  MoveL 5326 to (228.65, 164.04, 78.65) mm, rotated rx 180 ry 0 rz 180 deg; joints [-145.551, -82.193, -28.272, 62.992, 39.413, -56.586]
  Call Extruder(271.49953)
  MoveL 5327 to (228.4, 164.09, 78.65) mm, rotated rx 180 ry 0 rz 180 deg; joints [-145.535, -82.158, -28.345, 62.966, 39.444, -56.545]
  MoveL 5328 to (228.4, 164.09, 78.65) mm, rotated rx 180 ry 0 rz 180 deg; joints [-145.535, -82.158, -28.345, 62.966, 39.444, -56.545]
  Call Extruder(271.63590)
  MoveL 5329 to (228.15, 164.14, 78.65) mm, rotated rx -180 ry 0 rz 180 deg; joints [-145.518, -82.122, -28.418, 62.94, 39.475, -56.503]
  MoveL 5330 to (228.15, 164.14, 78.65) mm, rotated rx -180 ry 0 rz 180 deg; joints [-145.518, -82.122, -28.418, 62.94, 39.475, -56.503]
  Call Extruder(271.77166)
  MoveL 5331 to (227.9, 164.19, 78.65) mm, rotated rx 180 ry 0 rz 180 deg; joints [-145.502, -82.086, -28.49, 62.914, 39.505, -56.463]
  MoveL 5332 to (227.9, 164.19, 78.65) mm, rotated rx 180 ry 0 rz 180 deg; joints [-145.502, -82.086, -28.49, 62.914, 39.505, -56.463]
  Call Extruder(271.90680)
  MoveL 5333 to (227.65, 164.24, 78.65) mm, rotated rx 180 ry 0 rz -180 deg; joints [-145.485, -82.051, -28.563, 62.889, 39.536, -56.422]
  MoveL 5334 to (227.65, 164.24, 78.65) mm, rotated rx 180 ry 0 rz -180 deg; joints [-145.485, -82.051, -28.563, 62.889, 39.536, -56.422]
  Call Extruder(272.04134)
  MoveL 5335 to (227.4, 164.29, 78.65) mm, rotated rx 180 ry 0 rz 180 deg; joints [-145.469, -82.016, -28.635, 62.863, 39.566, -56.382]
  MoveL 5336 to (227.4, 164.29, 78.65) mm, rotated rx 180 ry 0 rz 180 deg; joints [-145.469, -82.016, -28.635, 62.863, 39.566, -56.382]
  Call Extruder(272.17527)
  MoveL 5337 to (227.15, 164.34, 78.65) mm, rotated rx 180 ry 0 rz -180 deg; joints [-145.453, -81.98, -28.707, 62.838, 39.597, -56.341]
  MoveL 5338 to (227.15, 164.34, 78.65) mm, rotated rx 180 ry 0 rz -180 deg; joints [-145.453, -81.98, -28.707, 62.838, 39.597, -56.341]
  Call Extruder(272.32313)
  MoveL 5339 to (226.87, 164.39, 78.65) mm, rotated rx 180 ry 0 rz -180 deg; joints [-145.435, -81.94, -28.788, 62.809, 39.63, -56.295]
  MoveL 5340 to (226.87, 164.39, 78.65) mm, rotated rx 180 ry 0 rz -180 deg; joints [-145.435, -81.94, -28.788, 62.809, 39.63, -56.295]
  Call Extruder(272.48487)
  MoveL 5341 to (226.57, 164.44, 78.65) mm, rotated rx 180 ry 0 rz 180 deg; joints [-145.415, -81.896, -28.879, 62.776, 39.668, -56.244]
  MoveL 5342 to (226.57, 164.44, 78.65) mm, rotated rx 180 ry 0 rz 180 deg; joints [-145.415, -81.896, -28.879, 62.776, 39.668, -56.244]
  Call Extruder(272.64589)
  MoveL 5343 to (226.26, 164.49, 78.65) mm, rotated rx 180 ry 0 rz -180 deg; joints [-145.396, -81.851, -28.97, 62.743, 39.705, -56.192]
  MoveL 5344 to (226.26, 164.49, 78.65) mm, rotated rx 180 ry 0 rz -180 deg; joints [-145.396, -81.851, -28.97, 62.743, 39.705, -56.192]
  Call Extruder(272.80617)
  MoveL 5345 to (225.96, 164.53, 78.65) mm, rotated rx 180 ry 0 rz 180 deg; joints [-145.377, -81.807, -29.061, 62.711, 39.742, -56.141]
  MoveL 5346 to (225.96, 164.53, 78.65) mm, rotated rx 180 ry 0 rz 180 deg; joints [-145.377, -81.807, -29.061, 62.711, 39.742, -56.141]
  Call Extruder(272.96573)
  MoveL 5347 to (225.65, 164.58, 78.65) mm, rotated rx 180 ry 0 rz 180 deg; joints [-145.357, -81.763, -29.151, 62.678, 39.779, -56.09]
  MoveL 5348 to (225.65, 164.58, 78.65) mm, rotated rx 180 ry 0 rz 180 deg; joints [-145.357, -81.763, -29.151, 62.678, 39.779, -56.09]
  Call Extruder(273.12456)
  MoveL 5349 to (225.34, 164.63, 78.65) mm, rotated rx -180 ry 0 rz 180 deg; joints [-145.338, -81.719, -29.241, 62.646, 39.817, -56.039]
  MoveL 5350 to (225.34, 164.63, 78.65) mm, rotated rx -180 ry 0 rz 180 deg; joints [-145.338, -81.719, -29.241, 62.646, 39.817, -56.039]
  Call Extruder(273.30323)
  MoveL 5351 to (225, 164.68, 78.65) mm, rotated rx -180 ry 0 rz 180 deg; joints [-145.317, -81.668, -29.344, 62.608, 39.859, -55.98]
  MoveL 5352 to (225, 164.68, 78.65) mm, rotated rx -180 ry 0 rz 180 deg; joints [-145.317, -81.668, -29.344, 62.608, 39.859, -55.98]
  Call Extruder(273.50167)
  MoveL 5353 to (224.61, 164.72, 78.65) mm, rotated rx 180 ry 0 rz 180 deg; joints [-145.293, -81.611, -29.461, 62.565, 39.906, -55.913]
  MoveL 5354 to (224.61, 164.72, 78.65) mm, rotated rx 180 ry 0 rz 180 deg; joints [-145.293, -81.611, -29.461, 62.565, 39.906, -55.913]
  Call Extruder(273.69925)
  MoveL 5355 to (224.22, 164.77, 78.65) mm, rotated rx 180 ry 0 rz 180 deg; joints [-145.27, -81.554, -29.578, 62.523, 39.953, -55.846]
  MoveL 5356 to (224.22, 164.77, 78.65) mm, rotated rx 180 ry 0 rz 180 deg; joints [-145.27, -81.554, -29.578, 62.523, 39.953, -55.846]
  Call Extruder(273.89595)
  MoveL 5357 to (223.83, 164.82, 78.65) mm, rotated rx -180 ry 0 rz 180 deg; joints [-145.246, -81.497, -29.694, 62.48, 39.999, -55.78]
  MoveL 5358 to (223.83, 164.82, 78.65) mm, rotated rx -180 ry 0 rz 180 deg; joints [-145.246, -81.497, -29.694, 62.48, 39.999, -55.78]
  Call Extruder(274.09179)
  MoveL 5359 to (223.45, 164.86, 78.65) mm, rotated rx -180 ry 0 rz 180 deg; joints [-145.223, -81.44, -29.811, 62.438, 40.046, -55.713]
  MoveL 5360 to (223.45, 164.86, 78.65) mm, rotated rx -180 ry 0 rz 180 deg; joints [-145.223, -81.44, -29.811, 62.438, 40.046, -55.713]
  Call Extruder(274.38715)
  MoveL 5361 to (222.86, 164.91, 78.65) mm, rotated rx 180 ry 0 rz 180 deg; joints [-145.189, -81.352, -29.991, 62.371, 40.117, -55.609]
  MoveL 5362 to (222.86, 164.91, 78.65) mm, rotated rx 180 ry 0 rz 180 deg; joints [-145.189, -81.352, -29.991, 62.371, 40.117, -55.609]
  Call Extruder(274.68118)
  MoveL 5363 to (222.27, 164.95, 78.65) mm, rotated rx 180 ry 0 rz -180 deg; joints [-145.155, -81.264, -30.172, 62.304, 40.188, -55.505]
  MoveL 5364 to (222.27, 164.95, 78.65) mm, rotated rx 180 ry 0 rz -180 deg; joints [-145.155, -81.264, -30.172, 62.304, 40.188, -55.505]
  Call Extruder(274.97387)
  MoveL 5365 to (221.68, 165, 78.65) mm, rotated rx 180 ry 0 rz -180 deg; joints [-145.121, -81.176, -30.351, 62.238, 40.259, -55.402]
  MoveL 5366 to (221.68, 165, 78.65) mm, rotated rx 180 ry 0 rz -180 deg; joints [-145.121, -81.176, -30.351, 62.238, 40.259, -55.402]
  Call Extruder(275.54732)
  MoveL 5367 to (220.52, 165.05, 78.65) mm, rotated rx -180 ry 0 rz -180 deg; joints [-145.056, -81, -30.712, 62.101, 40.398, -55.192]
  MoveL 5368 to (220.52, 165.05, 78.65) mm, rotated rx -180 ry 0 rz -180 deg; joints [-145.056, -81, -30.712, 62.101, 40.398, -55.192]
  Call Extruder(276.26133)
  MoveL 5369 to (219.06, 165.09, 78.65) mm, rotated rx 180 ry 0 rz -180 deg; joints [-144.977, -80.78, -31.164, 61.931, 40.572, -54.93]
  Call Extruder(393.10807)
  MoveL 5370 to (-19.06, 165.09, 78.65) mm, rotated rx 180 ry 0 rz 180 deg; joints [-127.435, -60.323, -76.536, 60.813, 65.44, -36.653]
  Call Extruder(393.53667)
  MoveL 5371 to (-19.94, 165.07, 78.65) mm, rotated rx 180 ry 0 rz 180 deg; joints [-127.348, -60.28, -76.645, 60.863, 65.523, -36.622]
  MoveL 5372 to (-19.94, 165.07, 78.65) mm, rotated rx 180 ry 0 rz 180 deg; joints [-127.348, -60.28, -76.645, 60.863, 65.523, -36.622]
  Call Extruder(394.11012)
  MoveL 5373 to (-21.1, 165.02, 78.65) mm, rotated rx 180 ry 0 rz -180 deg; joints [-127.235, -60.221, -76.793, 60.928, 65.634, -36.579]
  MoveL 5374 to (-21.1, 165.02, 78.65) mm, rotated rx 180 ry 0 rz -180 deg; joints [-127.235, -60.221, -76.793, 60.928, 65.634, -36.579]
  Call Extruder(394.54442)
  MoveL 5375 to (-21.97, 164.98, 78.65) mm, rotated rx 180 ry 0 rz -180 deg; joints [-127.15, -60.176, -76.906, 60.976, 65.718, -36.544]
  MoveL 5376 to (-21.97, 164.98, 78.65) mm, rotated rx 180 ry 0 rz -180 deg; joints [-127.15, -60.176, -76.906, 60.976, 65.718, -36.544]
  Call Extruder(394.83845)
  MoveL 5377 to (-22.56, 164.93, 78.65) mm, rotated rx 180 ry 0 rz 180 deg; joints [-127.093, -60.144, -76.984, 61.007, 65.774, -36.519]
  MoveL 5378 to (-22.56, 164.93, 78.65) mm, rotated rx 180 ry 0 rz 180 deg; joints [-127.093, -60.144, -76.984, 61.007, 65.774, -36.519]
  Call Extruder(395.13381)
  MoveL 5379 to (-23.15, 164.89, 78.65) mm, rotated rx -180 ry 0 rz -180 deg; joints [-127.037, -60.113, -77.062, 61.038, 65.83, -36.495]
  MoveL 5380 to (-23.15, 164.89, 78.65) mm, rotated rx -180 ry 0 rz -180 deg; joints [-127.037, -60.113, -77.062, 61.038, 65.83, -36.495]
  Call Extruder(395.38003)
  MoveL 5381 to (-23.64, 164.84, 78.65) mm, rotated rx 180 ry 0 rz 180 deg; joints [-126.991, -60.087, -77.128, 61.063, 65.877, -36.473]
  MoveL 5382 to (-23.64, 164.84, 78.65) mm, rotated rx 180 ry 0 rz 180 deg; joints [-126.991, -60.087, -77.128, 61.063, 65.877, -36.473]
  Call Extruder(395.57673)
  MoveL 5383 to (-24.03, 164.79, 78.65) mm, rotated rx 180 ry 0 rz 180 deg; joints [-126.955, -60.066, -77.181, 61.082, 65.914, -36.455]
  MoveL 5384 to (-24.03, 164.79, 78.65) mm, rotated rx 180 ry 0 rz 180 deg; joints [-126.955, -60.066, -77.181, 61.082, 65.914, -36.455]
  Call Extruder(395.77431)
  MoveL 5385 to (-24.42, 164.75, 78.65) mm, rotated rx 180 ry 0 rz 180 deg; joints [-126.919, -60.045, -77.235, 61.101, 65.951, -36.437]
  MoveL 5386 to (-24.42, 164.75, 78.65) mm, rotated rx 180 ry 0 rz 180 deg; joints [-126.919, -60.045, -77.235, 61.101, 65.951, -36.437]
  Call Extruder(395.97275)
  MoveL 5387 to (-24.8, 164.7, 78.65) mm, rotated rx -180 ry 0 rz 180 deg; joints [-126.883, -60.023, -77.289, 61.121, 65.988, -36.419]
  MoveL 5388 to (-24.8, 164.7, 78.65) mm, rotated rx -180 ry 0 rz 180 deg; joints [-126.883, -60.023, -77.289, 61.121, 65.988, -36.419]
  Call Extruder(396.17206)
  MoveL 5389 to (-25.19, 164.66, 78.65) mm, rotated rx 180 ry 0 rz -180 deg; joints [-126.847, -60.002, -77.342, 61.14, 66.025, -36.401]
  MoveL 5390 to (-25.19, 164.66, 78.65) mm, rotated rx 180 ry 0 rz -180 deg; joints [-126.847, -60.002, -77.342, 61.14, 66.025, -36.401]
  Call Extruder(396.33089)
  MoveL 5391 to (-25.5, 164.61, 78.65) mm, rotated rx 180 ry 0 rz 180 deg; joints [-126.82, -59.985, -77.386, 61.154, 66.054, -36.386]
  MoveL 5392 to (-25.5, 164.61, 78.65) mm, rotated rx 180 ry 0 rz 180 deg; joints [-126.82, -59.985, -77.386, 61.154, 66.054, -36.386]
  Call Extruder(396.49045)
  MoveL 5393 to (-25.8, 164.56, 78.65) mm, rotated rx -180 ry 0 rz 180 deg; joints [-126.792, -59.967, -77.43, 61.168, 66.083, -36.37]
  MoveL 5394 to (-25.8, 164.56, 78.65) mm, rotated rx -180 ry 0 rz 180 deg; joints [-126.792, -59.967, -77.43, 61.168, 66.083, -36.37]
  Call Extruder(396.65073)
  MoveL 5395 to (-26.11, 164.51, 78.65) mm, rotated rx 180 ry 0 rz 180 deg; joints [-126.765, -59.95, -77.474, 61.182, 66.112, -36.355]
  MoveL 5396 to (-26.11, 164.51, 78.65) mm, rotated rx 180 ry 0 rz 180 deg; joints [-126.765, -59.95, -77.474, 61.182, 66.112, -36.355]
  Call Extruder(396.81175)
  MoveL 5397 to (-26.41, 164.46, 78.65) mm, rotated rx -180 ry 0 rz -180 deg; joints [-126.737, -59.932, -77.518, 61.196, 66.141, -36.339]
  MoveL 5398 to (-26.41, 164.46, 78.65) mm, rotated rx -180 ry 0 rz -180 deg; joints [-126.737, -59.932, -77.518, 61.196, 66.141, -36.339]
  Call Extruder(396.97349)
  MoveL 5399 to (-26.72, 164.41, 78.65) mm, rotated rx -180 ry 0 rz 180 deg; joints [-126.71, -59.915, -77.562, 61.21, 66.17, -36.323]
  MoveL 5400 to (-26.72, 164.41, 78.65) mm, rotated rx -180 ry 0 rz 180 deg; joints [-126.71, -59.915, -77.562, 61.21, 66.17, -36.323]
  Call Extruder(397.13596)
  MoveL 5401 to (-27.03, 164.36, 78.65) mm, rotated rx -180 ry 0 rz 180 deg; joints [-126.682, -59.897, -77.606, 61.224, 66.199, -36.308]
  MoveL 5402 to (-27.03, 164.36, 78.65) mm, rotated rx -180 ry 0 rz 180 deg; joints [-126.682, -59.897, -77.606, 61.224, 66.199, -36.308]
  Call Extruder(397.26988)
  MoveL 5403 to (-27.27, 164.32, 78.65) mm, rotated rx 180 ry 0 rz -180 deg; joints [-126.66, -59.883, -77.643, 61.234, 66.223, -36.294]
  MoveL 5404 to (-27.27, 164.32, 78.65) mm, rotated rx 180 ry 0 rz -180 deg; joints [-126.66, -59.883, -77.643, 61.234, 66.223, -36.294]
  Call Extruder(397.40442)
  MoveL 5405 to (-27.52, 164.27, 78.65) mm, rotated rx 180 ry 0 rz -180 deg; joints [-126.638, -59.868, -77.68, 61.245, 66.247, -36.28]
  MoveL 5406 to (-27.52, 164.27, 78.65) mm, rotated rx 180 ry 0 rz -180 deg; joints [-126.638, -59.868, -77.68, 61.245, 66.247, -36.28]
  Call Extruder(397.53957)
  MoveL 5407 to (-27.77, 164.22, 78.65) mm, rotated rx -180 ry 0 rz 180 deg; joints [-126.617, -59.853, -77.718, 61.255, 66.271, -36.266]
  MoveL 5408 to (-27.77, 164.22, 78.65) mm, rotated rx -180 ry 0 rz 180 deg; joints [-126.617, -59.853, -77.718, 61.255, 66.271, -36.266]
  Call Extruder(397.67532)
  MoveL 5409 to (-28.02, 164.17, 78.65) mm, rotated rx -180 ry 0 rz -180 deg; joints [-126.595, -59.838, -77.755, 61.266, 66.294, -36.253]
  MoveL 5410 to (-28.02, 164.17, 78.65) mm, rotated rx -180 ry 0 rz -180 deg; joints [-126.595, -59.838, -77.755, 61.266, 66.294, -36.253]
  Call Extruder(397.81169)
  MoveL 5411 to (-28.27, 164.12, 78.65) mm, rotated rx 180 ry 0 rz 180 deg; joints [-126.573, -59.824, -77.792, 61.276, 66.318, -36.239]
  MoveL 5412 to (-28.27, 164.12, 78.65) mm, rotated rx 180 ry 0 rz 180 deg; joints [-126.573, -59.824, -77.792, 61.276, 66.318, -36.239]
  Call Extruder(397.89656)
  MoveL 5413 to (-28.42, 164.09, 78.65) mm, rotated rx 180 ry 0 rz 180 deg; joints [-126.559, -59.815, -77.815, 61.283, 66.333, -36.23]
  Set speed (130.0 mm/s)
  MoveL 5414 to (-31.76, 163.31, 78.65) mm, rotated rx 180 ry 0 rz 180 deg; joints [-126.274, -59.612, -78.328, 61.416, 66.65, -36.033]
  MoveL 5415 to (-31.76, 163.31, 88.06) mm, rotated rx 180 ry 0 rz 180 deg; joints [-126.274, -58.332, -78.939, 61.672, 66.331, -36.675]
  Call Extruder(395.89656)
  Set speed (40.0 mm/s)
  MoveL 5416 to (-31.76, 163.31, 88.06) mm, rotated rx 180 ry 0 rz 180 deg; joints [-126.274, -58.332, -78.939, 61.672, 66.331, -36.675]
  Call Extruder(0.00000)
  Set speed (130.0 mm/s)
  MoveL 5417 to (-31.64, 163.21, 88.06) mm, rotated rx 180 ry 0 rz 180 deg; joints [-126.294, -58.331, -78.941, 61.654, 66.319, -36.667]
  Call Extruder(2.00000)
  Set speed (40.0 mm/s)
  MoveL 5418 to (-31.64, 163.21, 88.06) mm, rotated rx 180 ry 0 rz 180 deg; joints [-126.294, -58.331, -78.941, 61.654, 66.319, -36.667]
  Set speed (30.0 mm/s)
  MoveL 5419 to (-31.64, 163.21, 88.06) mm, rotated rx 180 ry 0 rz 180 deg; joints [-126.294, -58.331, -78.941, 61.654, 66.319, -36.667]
  Call Extruder(2.18198)
  MoveL 5420 to (-31.93, 163.09, 88.06) mm, rotated rx -180 ry 0 rz 180 deg; joints [-126.273, -58.309, -78.994, 61.66, 66.347, -36.644]
  MoveL 5421 to (-31.93, 163.09, 88.06) mm, rotated rx -180 ry 0 rz 180 deg; joints [-126.273, -58.309, -78.994, 61.66, 66.347, -36.644]
  Call Extruder(2.36471)
  MoveL 5422 to (-32.22, 162.96, 88.06) mm, rotated rx -180 ry 0 rz 180 deg; joints [-126.252, -58.288, -79.047, 61.666, 66.375, -36.621]
  MoveL 5423 to (-32.22, 162.96, 88.06) mm, rotated rx -180 ry 0 rz 180 deg; joints [-126.252, -58.288, -79.047, 61.666, 66.375, -36.621]
  Call Extruder(2.53513)
  MoveL 5424 to (-32.49, 162.85, 88.06) mm, rotated rx 180 ry 0 rz 180 deg; joints [-126.233, -58.268, -79.097, 61.672, 66.4, -36.599]
  MoveL 5425 to (-32.49, 162.85, 88.06) mm, rotated rx 180 ry 0 rz 180 deg; joints [-126.233, -58.268, -79.097, 61.672, 66.4, -36.599]
  Call Extruder(2.69310)
  MoveL 5426 to (-32.74, 162.74, 88.06) mm, rotated rx 180 ry 0 rz 180 deg; joints [-126.215, -58.25, -79.142, 61.677, 66.424, -36.579]
  MoveL 5427 to (-32.74, 162.74, 88.06) mm, rotated rx 180 ry 0 rz 180 deg; joints [-126.215, -58.25, -79.142, 61.677, 66.424, -36.579]
  Call Extruder(2.85168)
  MoveL 5428 to (-32.99, 162.64, 88.06) mm, rotated rx 180 ry 0 rz -180 deg; joints [-126.197, -58.231, -79.188, 61.682, 66.448, -36.559]
  MoveL 5429 to (-32.99, 162.64, 88.06) mm, rotated rx 180 ry 0 rz -180 deg; joints [-126.197, -58.231, -79.188, 61.682, 66.448, -36.559]
  Call Extruder(3.05785)
  MoveL 5430 to (-33.29, 162.46, 88.06) mm, rotated rx 180 ry 0 rz 180 deg; joints [-126.179, -58.206, -79.251, 61.684, 66.476, -36.529]
  MoveL 5431 to (-33.29, 162.46, 88.06) mm, rotated rx 180 ry 0 rz 180 deg; joints [-126.179, -58.206, -79.251, 61.684, 66.476, -36.529]
  Call Extruder(3.26479)
  MoveL 5432 to (-33.6, 162.29, 88.06) mm, rotated rx 180 ry 0 rz 180 deg; joints [-126.16, -58.181, -79.314, 61.685, 66.505, -36.499]
  MoveL 5433 to (-33.6, 162.29, 88.06) mm, rotated rx 180 ry 0 rz 180 deg; joints [-126.16, -58.181, -79.314, 61.685, 66.505, -36.499]
  Call Extruder(3.47251)
  MoveL 5434 to (-33.9, 162.11, 88.06) mm, rotated rx 180 ry 0 rz 180 deg; joints [-126.142, -58.156, -79.377, 61.687, 66.534, -36.47]
  MoveL 5435 to (-33.9, 162.11, 88.06) mm, rotated rx 180 ry 0 rz 180 deg; joints [-126.142, -58.156, -79.377, 61.687, 66.534, -36.47]
  Call Extruder(3.68102)
  MoveL 5436 to (-34.21, 161.94, 88.06) mm, rotated rx 180 ry 0 rz 180 deg; joints [-126.123, -58.131, -79.44, 61.689, 66.563, -36.44]
  MoveL 5437 to (-34.21, 161.94, 88.06) mm, rotated rx 180 ry 0 rz 180 deg; joints [-126.123, -58.131, -79.44, 61.689, 66.563, -36.44]
  Call Extruder(3.86055)
  MoveL 5438 to (-34.45, 161.76, 88.06) mm, rotated rx 180 ry 0 rz 180 deg; joints [-126.111, -58.108, -79.496, 61.687, 66.586, -36.412]
  MoveL 5439 to (-34.45, 161.76, 88.06) mm, rotated rx 180 ry 0 rz 180 deg; joints [-126.111, -58.108, -79.496, 61.687, 66.586, -36.412]
  Call Extruder(4.19399)
  MoveL 5440 to (-34.9, 161.43, 88.06) mm, rotated rx 180 ry 0 rz -180 deg; joints [-126.089, -58.067, -79.6, 61.682, 66.629, -36.36]
  MoveL 5441 to (-34.9, 161.43, 88.06) mm, rotated rx 180 ry 0 rz -180 deg; joints [-126.089, -58.067, -79.6, 61.682, 66.629, -36.36]
  Call Extruder(4.52861)
  MoveL 5442 to (-35.35, 161.1, 88.06) mm, rotated rx -180 ry 0 rz 180 deg; joints [-126.067, -58.025, -79.703, 61.678, 66.672, -36.308]
  Call Extruder(5.35652)
  MoveL 5443 to (-36.39, 160.19, 88.06) mm, rotated rx 180 ry 0 rz 180 deg; joints [-126.027, -57.921, -79.966, 61.653, 66.77, -36.17]
  Call Extruder(6.18445)
  MoveL 5444 to (-37.3, 159.15, 88.06) mm, rotated rx 180 ry 0 rz 180 deg; joints [-126.011, -57.814, -80.233, 61.607, 66.856, -36.022]
  Call Extruder(6.35176)
  MoveL 5445 to (-37.47, 158.93, 88.06) mm, rotated rx -180 ry 0 rz 180 deg; joints [-126.011, -57.793, -80.288, 61.595, 66.872, -35.991]
  MoveL 5446 to (-37.47, 158.93, 88.06) mm, rotated rx -180 ry 0 rz 180 deg; joints [-126.011, -57.793, -80.288, 61.595, 66.872, -35.991]
  Call Extruder(6.68519)
  MoveL 5447 to (-37.79, 158.48, 88.06) mm, rotated rx -180 ry 0 rz 180 deg; joints [-126.011, -57.75, -80.396, 61.57, 66.903, -35.928]
  MoveL 5448 to (-37.79, 158.48, 88.06) mm, rotated rx -180 ry 0 rz 180 deg; joints [-126.011, -57.75, -80.396, 61.57, 66.903, -35.928]
  Call Extruder(7.01743)
  MoveL 5449 to (-38.12, 158.03, 88.06) mm, rotated rx 180 ry 0 rz 180 deg; joints [-126.011, -57.707, -80.504, 61.546, 66.934, -35.866]
  MoveL 5450 to (-38.12, 158.03, 88.06) mm, rotated rx 180 ry 0 rz 180 deg; joints [-126.011, -57.707, -80.504, 61.546, 66.934, -35.866]
  Call Extruder(7.13510)
  MoveL 5451 to (-38.22, 157.85, 88.06) mm, rotated rx -180 ry 0 rz 180 deg; joints [-126.013, -57.692, -80.542, 61.535, 66.943, -35.843]
  MoveL 5452 to (-38.22, 157.85, 88.06) mm, rotated rx -180 ry 0 rz 180 deg; joints [-126.013, -57.692, -80.542, 61.535, 66.943, -35.843]
  Call Extruder(7.34283)
  MoveL 5453 to (-38.4, 157.55, 88.06) mm, rotated rx -180 ry 0 rz -180 deg; joints [-126.018, -57.665, -80.61, 61.515, 66.96, -35.802]
  MoveL 5454 to (-38.4, 157.55, 88.06) mm, rotated rx -180 ry 0 rz -180 deg; joints [-126.018, -57.665, -80.61, 61.515, 66.96, -35.802]
  Call Extruder(7.54978)
  MoveL 5455 to (-38.57, 157.25, 88.06) mm, rotated rx 180 ry 0 rz 180 deg; joints [-126.023, -57.638, -80.677, 61.496, 66.976, -35.762]
  MoveL 5456 to (-38.57, 157.25, 88.06) mm, rotated rx 180 ry 0 rz 180 deg; joints [-126.023, -57.638, -80.677, 61.496, 66.976, -35.762]
  Call Extruder(7.75595)
  MoveL 5457 to (-38.75, 156.94, 88.06) mm, rotated rx -180 ry 0 rz 180 deg; joints [-126.028, -57.611, -80.745, 61.476, 66.993, -35.721]
  MoveL 5458 to (-38.75, 156.94, 88.06) mm, rotated rx -180 ry 0 rz 180 deg; joints [-126.028, -57.611, -80.745, 61.476, 66.993, -35.721]
  Call Extruder(7.93763)
  MoveL 5459 to (-38.89, 156.66, 88.06) mm, rotated rx -180 ry 0 rz 180 deg; joints [-126.034, -57.588, -80.804, 61.457, 67.006, -35.685]
  MoveL 5460 to (-38.89, 156.66, 88.06) mm, rotated rx -180 ry 0 rz 180 deg; joints [-126.034, -57.588, -80.804, 61.457, 67.006, -35.685]
  Call Extruder(8.09561)
  MoveL 5461 to (-39, 156.42, 88.06) mm, rotated rx -180 ry 0 rz 180 deg; joints [-126.042, -57.568, -80.855, 61.439, 67.017, -35.653]
  MoveL 5462 to (-39, 156.42, 88.06) mm, rotated rx -180 ry 0 rz 180 deg; joints [-126.042, -57.568, -80.855, 61.439, 67.017, -35.653]
  Call Extruder(8.25300)
  MoveL 5463 to (-39.1, 156.17, 88.06) mm, rotated rx -180 ry 0 rz -180 deg; joints [-126.05, -57.547, -80.906, 61.42, 67.027, -35.62]
  MoveL 5464 to (-39.1, 156.17, 88.06) mm, rotated rx -180 ry 0 rz -180 deg; joints [-126.05, -57.547, -80.906, 61.42, 67.027, -35.62]
  Call Extruder(8.43571)
  MoveL 5465 to (-39.23, 155.87, 88.06) mm, rotated rx -180 ry 0 rz -180 deg; joints [-126.06, -57.524, -80.966, 61.398, 67.038, -35.583]
  MoveL 5466 to (-39.23, 155.87, 88.06) mm, rotated rx -180 ry 0 rz -180 deg; joints [-126.06, -57.524, -80.966, 61.398, 67.038, -35.583]
  Call Extruder(8.61768)
  MoveL 5467 to (-39.35, 155.58, 88.06) mm, rotated rx -180 ry 0 rz 180 deg; joints [-126.07, -57.501, -81.025, 61.376, 67.05, -35.545]
  MoveL 5468 to (-39.35, 155.58, 88.06) mm, rotated rx -180 ry 0 rz 180 deg; joints [-126.07, -57.501, -81.025, 61.376, 67.05, -35.545]
  Call Extruder(8.76501)
  MoveL 5469 to (-39.44, 155.34, 88.06) mm, rotated rx 180 ry 0 rz 180 deg; joints [-126.079, -57.482, -81.073, 61.358, 67.058, -35.515]
  MoveL 5470 to (-39.44, 155.34, 88.06) mm, rotated rx 180 ry 0 rz 180 deg; joints [-126.079, -57.482, -81.073, 61.358, 67.058, -35.515]
  Call Extruder(8.87824)
  MoveL 5471 to (-39.5, 155.15, 88.06) mm, rotated rx -180 ry 0 rz 180 deg; joints [-126.087, -57.467, -81.109, 61.342, 67.064, -35.491]
  MoveL 5472 to (-39.5, 155.15, 88.06) mm, rotated rx -180 ry 0 rz 180 deg; joints [-126.087, -57.467, -81.109, 61.342, 67.064, -35.491]
  Call Extruder(8.99103)
  MoveL 5473 to (-39.56, 154.97, 88.06) mm, rotated rx -180 ry 0 rz 180 deg; joints [-126.095, -57.453, -81.145, 61.327, 67.07, -35.467]
  MoveL 5474 to (-39.56, 154.97, 88.06) mm, rotated rx -180 ry 0 rz 180 deg; joints [-126.095, -57.453, -81.145, 61.327, 67.07, -35.467]
  Call Extruder(9.10338)
  MoveL 5475 to (-39.62, 154.78, 88.06) mm, rotated rx -180 ry 0 rz 180 deg; joints [-126.103, -57.439, -81.182, 61.312, 67.076, -35.443]
  MoveL 5476 to (-39.62, 154.78, 88.06) mm, rotated rx -180 ry 0 rz 180 deg; joints [-126.103, -57.439, -81.182, 61.312, 67.076, -35.443]
  Call Extruder(9.21528)
  MoveL 5477 to (-39.68, 154.59, 88.06) mm, rotated rx 180 ry 0 rz 180 deg; joints [-126.111, -57.425, -81.218, 61.296, 67.082, -35.42]
  MoveL 5478 to (-39.68, 154.59, 88.06) mm, rotated rx 180 ry 0 rz 180 deg; joints [-126.111, -57.425, -81.218, 61.296, 67.082, -35.42]
  Call Extruder(9.33668)
  MoveL 5479 to (-39.75, 154.38, 88.06) mm, rotated rx -180 ry 0 rz 180 deg; joints [-126.12, -57.409, -81.257, 61.279, 67.088, -35.394]
  MoveL 5480 to (-39.75, 154.38, 88.06) mm, rotated rx -180 ry 0 rz 180 deg; joints [-126.12, -57.409, -81.257, 61.279, 67.088, -35.394]
  Call Extruder(9.46747)
  MoveL 5481 to (-39.82, 154.16, 88.06) mm, rotated rx -180 ry 0 rz 180 deg; joints [-126.131, -57.392, -81.3, 61.261, 67.094, -35.366]
  MoveL 5482 to (-39.82, 154.16, 88.06) mm, rotated rx -180 ry 0 rz 180 deg; joints [-126.131, -57.392, -81.3, 61.261, 67.094, -35.366]
  Call Extruder(9.59770)
  MoveL 5483 to (-39.88, 153.94, 88.06) mm, rotated rx 180 ry 0 rz -180 deg; joints [-126.141, -57.376, -81.342, 61.242, 67.101, -35.338]
  MoveL 5484 to (-39.88, 153.94, 88.06) mm, rotated rx 180 ry 0 rz -180 deg; joints [-126.141, -57.376, -81.342, 61.242, 67.101, -35.338]
  Call Extruder(9.72737)
  MoveL 5485 to (-39.95, 153.71, 88.06) mm, rotated rx 180 ry 0 rz 180 deg; joints [-126.151, -57.359, -81.384, 61.223, 67.107, -35.31]
  MoveL 5486 to (-39.95, 153.71, 88.06) mm, rotated rx 180 ry 0 rz 180 deg; joints [-126.151, -57.359, -81.384, 61.223, 67.107, -35.31]
  Call Extruder(9.85647)
  MoveL 5487 to (-40.02, 153.49, 88.06) mm, rotated rx 180 ry 0 rz -180 deg; joints [-126.161, -57.342, -81.427, 61.205, 67.113, -35.282]
  MoveL 5488 to (-40.02, 153.49, 88.06) mm, rotated rx 180 ry 0 rz -180 deg; joints [-126.161, -57.342, -81.427, 61.205, 67.113, -35.282]
  Call Extruder(9.97156)
  MoveL 5489 to (-40.06, 153.28, 88.06) mm, rotated rx -180 ry 0 rz 180 deg; joints [-126.173, -57.328, -81.463, 61.187, 67.118, -35.257]
  MoveL 5490 to (-40.06, 153.28, 88.06) mm, rotated rx -180 ry 0 rz 180 deg; joints [-126.173, -57.328, -81.463, 61.187, 67.118, -35.257]
  Call Extruder(10.08619)
  MoveL 5491 to (-40.11, 153.08, 88.06) mm, rotated rx 180 ry 0 rz 180 deg; joints [-126.184, -57.313, -81.5, 61.169, 67.122, -35.232]
  MoveL 5492 to (-40.11, 153.08, 88.06) mm, rotated rx 180 ry 0 rz 180 deg; joints [-126.184, -57.313, -81.5, 61.169, 67.122, -35.232]
  Call Extruder(10.20038)
  MoveL 5493 to (-40.15, 152.88, 88.06) mm, rotated rx 180 ry 0 rz 180 deg; joints [-126.195, -57.299, -81.537, 61.15, 67.126, -35.207]
  MoveL 5494 to (-40.15, 152.88, 88.06) mm, rotated rx 180 ry 0 rz 180 deg; joints [-126.195, -57.299, -81.537, 61.15, 67.126, -35.207]
  Call Extruder(10.31411)
  MoveL 5495 to (-40.2, 152.67, 88.06) mm, rotated rx 180 ry 0 rz 180 deg; joints [-126.206, -57.285, -81.574, 61.132, 67.13, -35.182]
  MoveL 5496 to (-40.2, 152.67, 88.06) mm, rotated rx 180 ry 0 rz 180 deg; joints [-126.206, -57.285, -81.574, 61.132, 67.13, -35.182]
  Call Extruder(10.43953)
  MoveL 5497 to (-40.24, 152.45, 88.06) mm, rotated rx 180 ry 0 rz 180 deg; joints [-126.219, -57.269, -81.614, 61.112, 67.135, -35.154]
  MoveL 5498 to (-40.24, 152.45, 88.06) mm, rotated rx 180 ry 0 rz 180 deg; joints [-126.219, -57.269, -81.614, 61.112, 67.135, -35.154]
  Call Extruder(10.57651)
  MoveL 5499 to (-40.29, 152.19, 88.06) mm, rotated rx -180 ry 0 rz 180 deg; joints [-126.233, -57.251, -81.658, 61.089, 67.14, -35.123]
  MoveL 5500 to (-40.29, 152.19, 88.06) mm, rotated rx -180 ry 0 rz 180 deg; joints [-126.233, -57.251, -81.658, 61.089, 67.14, -35.123]
  Call Extruder(10.71287)
  MoveL 5501 to (-40.34, 151.95, 88.06) mm, rotated rx 180 ry 0 rz 180 deg; joints [-126.248, -57.234, -81.702, 61.066, 67.144, -35.093]
  MoveL 5502 to (-40.34, 151.95, 88.06) mm, rotated rx 180 ry 0 rz 180 deg; joints [-126.248, -57.234, -81.702, 61.066, 67.144, -35.093]
  Call Extruder(10.84863)
  MoveL 5503 to (-40.39, 151.7, 88.06) mm, rotated rx 180 ry 0 rz 180 deg; joints [-126.262, -57.217, -81.746, 61.044, 67.149, -35.063]
  MoveL 5504 to (-40.39, 151.7, 88.06) mm, rotated rx 180 ry 0 rz 180 deg; joints [-126.262, -57.217, -81.746, 61.044, 67.149, -35.063]
  Call Extruder(10.98377)
  MoveL 5505 to (-40.44, 151.45, 88.06) mm, rotated rx -180 ry 0 rz 180 deg; joints [-126.276, -57.199, -81.79, 61.021, 67.154, -35.032]
  MoveL 5506 to (-40.44, 151.45, 88.06) mm, rotated rx -180 ry 0 rz 180 deg; joints [-126.276, -57.199, -81.79, 61.021, 67.154, -35.032]
  Call Extruder(11.11831)
  MoveL 5507 to (-40.49, 151.2, 88.06) mm, rotated rx -180 ry 0 rz -180 deg; joints [-126.291, -57.182, -81.834, 60.999, 67.159, -35.002]
  MoveL 5508 to (-40.49, 151.2, 88.06) mm, rotated rx -180 ry 0 rz -180 deg; joints [-126.291, -57.182, -81.834, 60.999, 67.159, -35.002]
  Call Extruder(11.25223)
  MoveL 5509 to (-40.54, 150.95, 88.06) mm, rotated rx 180 ry 0 rz 180 deg; joints [-126.305, -57.165, -81.878, 60.976, 67.163, -34.972]
  MoveL 5510 to (-40.54, 150.95, 88.06) mm, rotated rx 180 ry 0 rz 180 deg; joints [-126.305, -57.165, -81.878, 60.976, 67.163, -34.972]
  Call Extruder(11.40009)
  MoveL 5511 to (-40.59, 150.67, 88.06) mm, rotated rx -180 ry 0 rz 180 deg; joints [-126.322, -57.146, -81.927, 60.95, 67.168, -34.938]
  MoveL 5512 to (-40.59, 150.67, 88.06) mm, rotated rx -180 ry 0 rz 180 deg; joints [-126.322, -57.146, -81.927, 60.95, 67.168, -34.938]
  Call Extruder(11.56181)
  MoveL 5513 to (-40.64, 150.37, 88.06) mm, rotated rx -180 ry 0 rz -180 deg; joints [-126.341, -57.125, -81.979, 60.922, 67.173, -34.901]
  MoveL 5514 to (-40.64, 150.37, 88.06) mm, rotated rx -180 ry 0 rz -180 deg; joints [-126.341, -57.125, -81.979, 60.922, 67.173, -34.901]
  Call Extruder(11.72281)
  MoveL 5515 to (-40.69, 150.06, 88.06) mm, rotated rx -180 ry 0 rz 180 deg; joints [-126.36, -57.105, -82.032, 60.893, 67.178, -34.864]
  MoveL 5516 to (-40.69, 150.06, 88.06) mm, rotated rx -180 ry 0 rz 180 deg; joints [-126.36, -57.105, -82.032, 60.893, 67.178, -34.864]
  Call Extruder(11.88308)
  MoveL 5517 to (-40.73, 149.76, 88.06) mm, rotated rx 180 ry 0 rz 180 deg; joints [-126.379, -57.084, -82.084, 60.864, 67.182, -34.827]
  MoveL 5518 to (-40.73, 149.76, 88.06) mm, rotated rx 180 ry 0 rz 180 deg; joints [-126.379, -57.084, -82.084, 60.864, 67.182, -34.827]
  Call Extruder(12.04262)
  MoveL 5519 to (-40.78, 149.45, 88.06) mm, rotated rx 180 ry 0 rz -180 deg; joints [-126.398, -57.064, -82.137, 60.836, 67.187, -34.79]
  MoveL 5520 to (-40.78, 149.45, 88.06) mm, rotated rx 180 ry 0 rz -180 deg; joints [-126.398, -57.064, -82.137, 60.836, 67.187, -34.79]
  Call Extruder(12.20144)
  MoveL 5521 to (-40.83, 149.14, 88.06) mm, rotated rx 180 ry 0 rz 180 deg; joints [-126.417, -57.043, -82.189, 60.807, 67.192, -34.754]
  MoveL 5522 to (-40.83, 149.14, 88.06) mm, rotated rx 180 ry 0 rz 180 deg; joints [-126.417, -57.043, -82.189, 60.807, 67.192, -34.754]
  Call Extruder(12.38010)
  MoveL 5523 to (-40.88, 148.8, 88.06) mm, rotated rx 180 ry 0 rz 180 deg; joints [-126.439, -57.02, -82.248, 60.774, 67.196, -34.712]
  MoveL 5524 to (-40.88, 148.8, 88.06) mm, rotated rx 180 ry 0 rz 180 deg; joints [-126.439, -57.02, -82.248, 60.774, 67.196, -34.712]
  Call Extruder(12.57854)
  MoveL 5525 to (-40.92, 148.41, 88.06) mm, rotated rx 180 ry 0 rz 180 deg; joints [-126.465, -56.995, -82.313, 60.736, 67.201, -34.666]
  MoveL 5526 to (-40.92, 148.41, 88.06) mm, rotated rx 180 ry 0 rz 180 deg; joints [-126.465, -56.995, -82.313, 60.736, 67.201, -34.666]
  Call Extruder(12.77611)
  MoveL 5527 to (-40.97, 148.02, 88.06) mm, rotated rx 180 ry 0 rz 180 deg; joints [-126.491, -56.97, -82.377, 60.699, 67.205, -34.62]
  MoveL 5528 to (-40.97, 148.02, 88.06) mm, rotated rx 180 ry 0 rz 180 deg; joints [-126.491, -56.97, -82.377, 60.699, 67.205, -34.62]
  Call Extruder(12.97282)
  MoveL 5529 to (-41.02, 147.63, 88.06) mm, rotated rx 180 ry 0 rz -180 deg; joints [-126.517, -56.945, -82.442, 60.661, 67.21, -34.573]
  MoveL 5530 to (-41.02, 147.63, 88.06) mm, rotated rx 180 ry 0 rz -180 deg; joints [-126.517, -56.945, -82.442, 60.661, 67.21, -34.573]
  Call Extruder(13.16866)
  MoveL 5531 to (-41.06, 147.25, 88.06) mm, rotated rx 180 ry 0 rz -180 deg; joints [-126.543, -56.92, -82.506, 60.623, 67.214, -34.527]
  MoveL 5532 to (-41.06, 147.25, 88.06) mm, rotated rx 180 ry 0 rz -180 deg; joints [-126.543, -56.92, -82.506, 60.623, 67.214, -34.527]
  Call Extruder(13.46406)
  MoveL 5533 to (-41.11, 146.66, 88.06) mm, rotated rx 180 ry 0 rz -180 deg; joints [-126.585, -56.883, -82.601, 60.564, 67.219, -34.457]
  MoveL 5534 to (-41.11, 146.66, 88.06) mm, rotated rx 180 ry 0 rz -180 deg; joints [-126.585, -56.883, -82.601, 60.564, 67.219, -34.457]
  Call Extruder(13.75812)
  MoveL 5535 to (-41.15, 146.07, 88.06) mm, rotated rx 180 ry 0 rz -180 deg; joints [-126.628, -56.846, -82.696, 60.505, 67.224, -34.388]
  MoveL 5536 to (-41.15, 146.07, 88.06) mm, rotated rx 180 ry 0 rz -180 deg; joints [-126.628, -56.846, -82.696, 60.505, 67.224, -34.388]
  Call Extruder(14.05085)
  MoveL 5537 to (-41.2, 145.48, 88.06) mm, rotated rx 180 ry 0 rz 180 deg; joints [-126.67, -56.809, -82.792, 60.446, 67.228, -34.318]
  MoveL 5538 to (-41.2, 145.48, 88.06) mm, rotated rx 180 ry 0 rz 180 deg; joints [-126.67, -56.809, -82.792, 60.446, 67.228, -34.318]
  Call Extruder(14.62431)
  MoveL 5539 to (-41.25, 144.32, 88.06) mm, rotated rx 180 ry 0 rz 180 deg; joints [-126.759, -56.738, -82.973, 60.326, 67.233, -34.182]
  MoveL 5540 to (-41.25, 144.32, 88.06) mm, rotated rx 180 ry 0 rz 180 deg; joints [-126.759, -56.738, -82.973, 60.326, 67.233, -34.182]
  Call Extruder(15.33827)
  MoveL 5541 to (-41.29, 142.86, 88.06) mm, rotated rx 180 ry 0 rz 180 deg; joints [-126.873, -56.651, -83.198, 60.173, 67.238, -34.013]
  Call Extruder(57.40309)
  MoveL 5542 to (-41.29, 57.14, 88.06) mm, rotated rx -180 ry 0 rz 180 deg; joints [-135.148, -52.441, -94.861, 49.773, 67.482, -24.359]
  Call Extruder(57.83165)
  MoveL 5543 to (-41.27, 56.26, 88.06) mm, rotated rx 180 ry 0 rz -180 deg; joints [-135.25, -52.407, -94.964, 49.651, 67.485, -24.263]
  MoveL 5544 to (-41.27, 56.26, 88.06) mm, rotated rx 180 ry 0 rz -180 deg; joints [-135.25, -52.407, -94.964, 49.651, 67.485, -24.263]
  Call Extruder(58.40510)
  MoveL 5545 to (-41.23, 55.1, 88.06) mm, rotated rx -180 ry 0 rz 180 deg; joints [-135.387, -52.362, -95.099, 49.486, 67.487, -24.137]
  MoveL 5546 to (-41.23, 55.1, 88.06) mm, rotated rx -180 ry 0 rz 180 deg; joints [-135.387, -52.362, -95.099, 49.486, 67.487, -24.137]
  Call Extruder(58.83942)
  MoveL 5547 to (-41.18, 54.23, 88.06) mm, rotated rx -180 ry 0 rz 180 deg; joints [-135.493, -52.33, -95.198, 49.36, 67.487, -24.042]
  MoveL 5548 to (-41.18, 54.23, 88.06) mm, rotated rx -180 ry 0 rz 180 deg; joints [-135.493, -52.33, -95.198, 49.36, 67.487, -24.042]
  Call Extruder(59.13348)
  MoveL 5549 to (-41.13, 53.64, 88.06) mm, rotated rx 180 ry 0 rz 180 deg; joints [-135.566, -52.308, -95.263, 49.274, 67.486, -23.978]
  MoveL 5550 to (-41.13, 53.64, 88.06) mm, rotated rx 180 ry 0 rz 180 deg; joints [-135.566, -52.308, -95.263, 49.274, 67.486, -23.978]
  Call Extruder(59.42888)
  MoveL 5551 to (-41.09, 53.05, 88.06) mm, rotated rx 180 ry 0 rz 180 deg; joints [-135.64, -52.287, -95.328, 49.188, 67.484, -23.915]
  MoveL 5552 to (-41.09, 53.05, 88.06) mm, rotated rx 180 ry 0 rz 180 deg; joints [-135.64, -52.287, -95.328, 49.188, 67.484, -23.915]
  Call Extruder(59.67512)
  MoveL 5553 to (-41.04, 52.56, 88.06) mm, rotated rx 180 ry 0 rz 180 deg; joints [-135.701, -52.27, -95.38, 49.116, 67.483, -23.863]
  MoveL 5554 to (-41.04, 52.56, 88.06) mm, rotated rx 180 ry 0 rz 180 deg; joints [-135.701, -52.27, -95.38, 49.116, 67.483, -23.863]
  Call Extruder(59.87182)
  MoveL 5555 to (-40.99, 52.17, 88.06) mm, rotated rx 180 ry 0 rz 180 deg; joints [-135.751, -52.256, -95.421, 49.058, 67.48, -23.821]
  MoveL 5556 to (-40.99, 52.17, 88.06) mm, rotated rx 180 ry 0 rz 180 deg; joints [-135.751, -52.256, -95.421, 49.058, 67.48, -23.821]
  Call Extruder(60.06940)
  MoveL 5557 to (-40.95, 51.78, 88.06) mm, rotated rx 180 ry 0 rz -180 deg; joints [-135.801, -52.243, -95.462, 49, 67.478, -23.78]
  MoveL 5558 to (-40.95, 51.78, 88.06) mm, rotated rx 180 ry 0 rz -180 deg; joints [-135.801, -52.243, -95.462, 49, 67.478, -23.78]
  Call Extruder(60.26784)
  MoveL 5559 to (-40.9, 51.4, 88.06) mm, rotated rx -180 ry 0 rz -180 deg; joints [-135.852, -52.23, -95.502, 48.942, 67.475, -23.739]
  MoveL 5560 to (-40.9, 51.4, 88.06) mm, rotated rx -180 ry 0 rz -180 deg; joints [-135.852, -52.23, -95.502, 48.942, 67.475, -23.739]
  Call Extruder(60.46715)
  MoveL 5561 to (-40.86, 51.01, 88.06) mm, rotated rx 180 ry 0 rz 180 deg; joints [-135.902, -52.217, -95.542, 48.883, 67.473, -23.698]
  MoveL 5562 to (-40.86, 51.01, 88.06) mm, rotated rx 180 ry 0 rz 180 deg; joints [-135.902, -52.217, -95.542, 48.883, 67.473, -23.698]
  Call Extruder(60.62596)
  MoveL 5563 to (-40.81, 50.7, 88.06) mm, rotated rx -180 ry 0 rz -180 deg; joints [-135.943, -52.207, -95.573, 48.836, 67.47, -23.665]
  MoveL 5564 to (-40.81, 50.7, 88.06) mm, rotated rx -180 ry 0 rz -180 deg; joints [-135.943, -52.207, -95.573, 48.836, 67.47, -23.665]
  Call Extruder(60.78551)
  MoveL 5565 to (-40.76, 50.4, 88.06) mm, rotated rx 180 ry 0 rz -180 deg; joints [-135.984, -52.197, -95.603, 48.789, 67.467, -23.633]
  MoveL 5566 to (-40.76, 50.4, 88.06) mm, rotated rx 180 ry 0 rz -180 deg; joints [-135.984, -52.197, -95.603, 48.789, 67.467, -23.633]
  Call Extruder(60.94578)
  MoveL 5567 to (-40.71, 50.09, 88.06) mm, rotated rx -180 ry 0 rz 180 deg; joints [-136.025, -52.187, -95.633, 48.742, 67.464, -23.601]
  MoveL 5568 to (-40.71, 50.09, 88.06) mm, rotated rx -180 ry 0 rz 180 deg; joints [-136.025, -52.187, -95.633, 48.742, 67.464, -23.601]
  Call Extruder(61.10677)
  MoveL 5569 to (-40.66, 49.79, 88.06) mm, rotated rx 180 ry 0 rz -180 deg; joints [-136.067, -52.177, -95.663, 48.695, 67.461, -23.569]
  MoveL 5570 to (-40.66, 49.79, 88.06) mm, rotated rx 180 ry 0 rz -180 deg; joints [-136.067, -52.177, -95.663, 48.695, 67.461, -23.569]
  Call Extruder(61.26850)
  MoveL 5571 to (-40.61, 49.48, 88.06) mm, rotated rx 180 ry 0 rz -180 deg; joints [-136.108, -52.167, -95.694, 48.647, 67.458, -23.536]
  MoveL 5572 to (-40.61, 49.48, 88.06) mm, rotated rx 180 ry 0 rz -180 deg; joints [-136.108, -52.167, -95.694, 48.647, 67.458, -23.536]
  Call Extruder(61.43095)
  MoveL 5573 to (-40.56, 49.17, 88.06) mm, rotated rx -180 ry 0 rz 180 deg; joints [-136.149, -52.158, -95.724, 48.6, 67.455, -23.504]
  MoveL 5574 to (-40.56, 49.17, 88.06) mm, rotated rx -180 ry 0 rz 180 deg; joints [-136.149, -52.158, -95.724, 48.6, 67.455, -23.504]
  Call Extruder(61.56488)
  MoveL 5575 to (-40.52, 48.93, 88.06) mm, rotated rx 180 ry 0 rz 180 deg; joints [-136.184, -52.15, -95.747, 48.56, 67.451, -23.478]
  MoveL 5576 to (-40.52, 48.93, 88.06) mm, rotated rx 180 ry 0 rz 180 deg; joints [-136.184, -52.15, -95.747, 48.56, 67.451, -23.478]
  Call Extruder(61.69941)
  MoveL 5577 to (-40.47, 48.68, 88.06) mm, rotated rx 180 ry 0 rz 180 deg; joints [-136.219, -52.143, -95.77, 48.521, 67.448, -23.452]
  MoveL 5578 to (-40.47, 48.68, 88.06) mm, rotated rx 180 ry 0 rz 180 deg; joints [-136.219, -52.143, -95.77, 48.521, 67.448, -23.452]
  Call Extruder(61.83456)
  MoveL 5579 to (-40.42, 48.43, 88.06) mm, rotated rx -180 ry 0 rz -180 deg; joints [-136.254, -52.135, -95.793, 48.481, 67.444, -23.426]
  MoveL 5580 to (-40.42, 48.43, 88.06) mm, rotated rx -180 ry 0 rz -180 deg; joints [-136.254, -52.135, -95.793, 48.481, 67.444, -23.426]
  Call Extruder(61.97031)
  MoveL 5581 to (-40.37, 48.18, 88.06) mm, rotated rx 180 ry 0 rz 180 deg; joints [-136.288, -52.127, -95.817, 48.442, 67.441, -23.4]
  MoveL 5582 to (-40.37, 48.18, 88.06) mm, rotated rx 180 ry 0 rz 180 deg; joints [-136.288, -52.127, -95.817, 48.442, 67.441, -23.4]
  Call Extruder(62.10668)
  MoveL 5583 to (-40.32, 47.93, 88.06) mm, rotated rx 180 ry 0 rz 180 deg; joints [-136.323, -52.12, -95.84, 48.402, 67.437, -23.374]
  MoveL 5584 to (-40.32, 47.93, 88.06) mm, rotated rx 180 ry 0 rz 180 deg; joints [-136.323, -52.12, -95.84, 48.402, 67.437, -23.374]
  Call Extruder(62.24365)
  MoveL 5585 to (-40.27, 47.68, 88.06) mm, rotated rx 180 ry 0 rz 180 deg; joints [-136.358, -52.112, -95.863, 48.363, 67.434, -23.348]
  MoveL 5586 to (-40.27, 47.68, 88.06) mm, rotated rx 180 ry 0 rz 180 deg; joints [-136.358, -52.112, -95.863, 48.363, 67.434, -23.348]
  Call Extruder(62.38124)
  MoveL 5587 to (-40.22, 47.43, 88.06) mm, rotated rx 180 ry 0 rz 180 deg; joints [-136.393, -52.105, -95.886, 48.323, 67.43, -23.322]
  MoveL 5588 to (-40.22, 47.43, 88.06) mm, rotated rx 180 ry 0 rz 180 deg; joints [-136.393, -52.105, -95.886, 48.323, 67.43, -23.322]
  Call Extruder(62.49497)
  MoveL 5589 to (-40.17, 47.23, 88.06) mm, rotated rx -180 ry 0 rz -180 deg; joints [-136.422, -52.099, -95.905, 48.29, 67.427, -23.301]
  MoveL 5590 to (-40.17, 47.23, 88.06) mm, rotated rx -180 ry 0 rz -180 deg; joints [-136.422, -52.099, -95.905, 48.29, 67.427, -23.301]
  Call Extruder(62.60915)
  MoveL 5591 to (-40.13, 47.02, 88.06) mm, rotated rx 180 ry 0 rz 180 deg; joints [-136.452, -52.093, -95.923, 48.257, 67.424, -23.28]
  MoveL 5592 to (-40.13, 47.02, 88.06) mm, rotated rx 180 ry 0 rz 180 deg; joints [-136.452, -52.093, -95.923, 48.257, 67.424, -23.28]
  Call Extruder(62.72378)
  MoveL 5593 to (-40.08, 46.82, 88.06) mm, rotated rx -180 ry 0 rz 180 deg; joints [-136.481, -52.087, -95.941, 48.225, 67.421, -23.259]
  MoveL 5594 to (-40.08, 46.82, 88.06) mm, rotated rx -180 ry 0 rz 180 deg; joints [-136.481, -52.087, -95.941, 48.225, 67.421, -23.259]
  Call Extruder(62.83887)
  MoveL 5595 to (-40.04, 46.61, 88.06) mm, rotated rx 180 ry 0 rz -180 deg; joints [-136.51, -52.081, -95.96, 48.192, 67.417, -23.237]
  MoveL 5596 to (-40.04, 46.61, 88.06) mm, rotated rx 180 ry 0 rz -180 deg; joints [-136.51, -52.081, -95.96, 48.192, 67.417, -23.237]
  Call Extruder(62.96111)
  MoveL 5597 to (-39.98, 46.4, 88.06) mm, rotated rx 180 ry 0 rz 180 deg; joints [-136.542, -52.075, -95.978, 48.156, 67.413, -23.215]
  MoveL 5598 to (-39.98, 46.4, 88.06) mm, rotated rx 180 ry 0 rz 180 deg; joints [-136.542, -52.075, -95.978, 48.156, 67.413, -23.215]
  Call Extruder(63.09077)
  MoveL 5599 to (-39.92, 46.18, 88.06) mm, rotated rx 180 ry 0 rz 180 deg; joints [-136.576, -52.069, -95.996, 48.119, 67.408, -23.193]
  MoveL 5600 to (-39.92, 46.18, 88.06) mm, rotated rx 180 ry 0 rz 180 deg; joints [-136.576, -52.069, -95.996, 48.119, 67.408, -23.193]
  Call Extruder(63.22100)
  MoveL 5601 to (-39.85, 45.95, 88.06) mm, rotated rx 180 ry 0 rz -180 deg; joints [-136.61, -52.064, -96.013, 48.081, 67.402, -23.17]
  MoveL 5602 to (-39.85, 45.95, 88.06) mm, rotated rx 180 ry 0 rz -180 deg; joints [-136.61, -52.064, -96.013, 48.081, 67.402, -23.17]
  Call Extruder(63.35179)
  MoveL 5603 to (-39.78, 45.73, 88.06) mm, rotated rx 180 ry 0 rz 180 deg; joints [-136.644, -52.058, -96.031, 48.043, 67.397, -23.147]
  MoveL 5604 to (-39.78, 45.73, 88.06) mm, rotated rx 180 ry 0 rz 180 deg; joints [-136.644, -52.058, -96.031, 48.043, 67.397, -23.147]
  Call Extruder(63.48315)
  MoveL 5605 to (-39.71, 45.5, 88.06) mm, rotated rx 180 ry 0 rz 180 deg; joints [-136.678, -52.052, -96.049, 48.005, 67.391, -23.124]
  MoveL 5606 to (-39.71, 45.5, 88.06) mm, rotated rx 180 ry 0 rz 180 deg; joints [-136.678, -52.052, -96.049, 48.005, 67.391, -23.124]
  Call Extruder(63.59505)
  MoveL 5607 to (-39.65, 45.32, 88.06) mm, rotated rx 180 ry 0 rz -180 deg; joints [-136.707, -52.048, -96.063, 47.973, 67.386, -23.105]
  MoveL 5608 to (-39.65, 45.32, 88.06) mm, rotated rx 180 ry 0 rz -180 deg; joints [-136.707, -52.048, -96.063, 47.973, 67.386, -23.105]
  Call Extruder(63.70740)
  MoveL 5609 to (-39.59, 45.13, 88.06) mm, rotated rx 180 ry 0 rz 180 deg; joints [-136.737, -52.043, -96.078, 47.941, 67.381, -23.086]
  MoveL 5610 to (-39.59, 45.13, 88.06) mm, rotated rx 180 ry 0 rz 180 deg; joints [-136.737, -52.043, -96.078, 47.941, 67.381, -23.086]
  Call Extruder(63.82019)
  MoveL 5611 to (-39.53, 44.94, 88.06) mm, rotated rx -180 ry 0 rz 180 deg; joints [-136.766, -52.038, -96.092, 47.909, 67.376, -23.067]
  MoveL 5612 to (-39.53, 44.94, 88.06) mm, rotated rx -180 ry 0 rz 180 deg; joints [-136.766, -52.038, -96.092, 47.909, 67.376, -23.067]
  Call Extruder(63.93342)
  MoveL 5613 to (-39.47, 44.75, 88.06) mm, rotated rx -180 ry 0 rz -180 deg; joints [-136.796, -52.034, -96.106, 47.877, 67.371, -23.048]
  MoveL 5614 to (-39.47, 44.75, 88.06) mm, rotated rx -180 ry 0 rz -180 deg; joints [-136.796, -52.034, -96.106, 47.877, 67.371, -23.048]
  Call Extruder(64.04710)
  MoveL 5615 to (-39.41, 44.56, 88.06) mm, rotated rx -180 ry 0 rz 180 deg; joints [-136.825, -52.029, -96.121, 47.844, 67.366, -23.029]
  MoveL 5616 to (-39.41, 44.56, 88.06) mm, rotated rx -180 ry 0 rz 180 deg; joints [-136.825, -52.029, -96.121, 47.844, 67.366, -23.029]
  Call Extruder(64.22906)
  MoveL 5617 to (-39.29, 44.27, 88.06) mm, rotated rx 180 ry 0 rz -180 deg; joints [-136.873, -52.023, -96.14, 47.792, 67.356, -23]
  MoveL 5618 to (-39.29, 44.27, 88.06) mm, rotated rx 180 ry 0 rz -180 deg; joints [-136.873, -52.023, -96.14, 47.792, 67.356, -23]
  Call Extruder(64.41178)
  MoveL 5619 to (-39.16, 43.98, 88.06) mm, rotated rx 180 ry 0 rz -180 deg; joints [-136.922, -52.017, -96.158, 47.74, 67.346, -22.971]
  MoveL 5620 to (-39.16, 43.98, 88.06) mm, rotated rx 180 ry 0 rz -180 deg; joints [-136.922, -52.017, -96.158, 47.74, 67.346, -22.971]
  Call Extruder(64.58219)
  MoveL 5621 to (-39.05, 43.71, 88.06) mm, rotated rx 180 ry 0 rz 180 deg; joints [-136.967, -52.011, -96.176, 47.691, 67.336, -22.945]
  MoveL 5622 to (-39.05, 43.71, 88.06) mm, rotated rx 180 ry 0 rz 180 deg; joints [-136.967, -52.011, -96.176, 47.691, 67.336, -22.945]
  Call Extruder(64.74018)
  MoveL 5623 to (-38.94, 43.46, 88.06) mm, rotated rx -180 ry 0 rz 180 deg; joints [-137.009, -52.006, -96.191, 47.646, 67.327, -22.92]
  MoveL 5624 to (-38.94, 43.46, 88.06) mm, rotated rx -180 ry 0 rz 180 deg; joints [-137.009, -52.006, -96.191, 47.646, 67.327, -22.92]
  Call Extruder(64.89877)
  MoveL 5625 to (-38.84, 43.21, 88.06) mm, rotated rx -180 ry 0 rz 180 deg; joints [-137.05, -52.001, -96.207, 47.601, 67.318, -22.896]
  MoveL 5626 to (-38.84, 43.21, 88.06) mm, rotated rx -180 ry 0 rz 180 deg; joints [-137.05, -52.001, -96.207, 47.601, 67.318, -22.896]
  Call Extruder(65.10493)
  MoveL 5627 to (-38.66, 42.91, 88.06) mm, rotated rx 180 ry 0 rz -180 deg; joints [-137.107, -51.997, -96.22, 47.542, 67.302, -22.867]
  MoveL 5628 to (-38.66, 42.91, 88.06) mm, rotated rx 180 ry 0 rz -180 deg; joints [-137.107, -51.997, -96.22, 47.542, 67.302, -22.867]
  Call Extruder(65.31188)
  MoveL 5629 to (-38.49, 42.6, 88.06) mm, rotated rx 180 ry 0 rz -180 deg; joints [-137.163, -51.993, -96.233, 47.484, 67.286, -22.838]
  MoveL 5630 to (-38.49, 42.6, 88.06) mm, rotated rx 180 ry 0 rz -180 deg; joints [-137.163, -51.993, -96.233, 47.484, 67.286, -22.838]
  Call Extruder(65.51960)
  MoveL 5631 to (-38.31, 42.3, 88.06) mm, rotated rx 180 ry 0 rz -180 deg; joints [-137.219, -51.988, -96.247, 47.425, 67.271, -22.809]
  MoveL 5632 to (-38.31, 42.3, 88.06) mm, rotated rx 180 ry 0 rz -180 deg; joints [-137.219, -51.988, -96.247, 47.425, 67.271, -22.809]
  Call Extruder(65.72810)
  MoveL 5633 to (-38.13, 41.99, 88.06) mm, rotated rx 180 ry 0 rz 180 deg; joints [-137.275, -51.984, -96.26, 47.366, 67.255, -22.78]
  MoveL 5634 to (-38.13, 41.99, 88.06) mm, rotated rx 180 ry 0 rz 180 deg; joints [-137.275, -51.984, -96.26, 47.366, 67.255, -22.78]
  Call Extruder(65.90765)
  MoveL 5635 to (-37.96, 41.75, 88.06) mm, rotated rx -180 ry 0 rz 180 deg; joints [-137.324, -51.982, -96.266, 47.315, 67.239, -22.758]
  MoveL 5636 to (-37.96, 41.75, 88.06) mm, rotated rx -180 ry 0 rz 180 deg; joints [-137.324, -51.982, -96.266, 47.315, 67.239, -22.758]
  Call Extruder(66.24109)
  MoveL 5637 to (-37.63, 41.3, 88.06) mm, rotated rx 180 ry 0 rz -180 deg; joints [-137.415, -51.979, -96.277, 47.222, 67.208, -22.717]
  MoveL 5638 to (-37.63, 41.3, 88.06) mm, rotated rx 180 ry 0 rz -180 deg; joints [-137.415, -51.979, -96.277, 47.222, 67.208, -22.717]
  Call Extruder(66.57571)
  MoveL 5639 to (-37.3, 40.85, 88.06) mm, rotated rx 180 ry 0 rz -180 deg; joints [-137.506, -51.975, -96.288, 47.129, 67.178, -22.676]
  Call Extruder(67.40364)
  MoveL 5640 to (-36.39, 39.81, 88.06) mm, rotated rx 180 ry 0 rz -180 deg; joints [-137.733, -51.974, -96.292, 46.901, 67.093, -22.585]
  Call Extruder(68.23155)
  MoveL 5641 to (-35.35, 38.9, 88.06) mm, rotated rx 180 ry 0 rz -180 deg; joints [-137.958, -51.982, -96.265, 46.68, 66.994, -22.511]
  Call Extruder(68.39886)
  MoveL 5642 to (-35.13, 38.73, 88.06) mm, rotated rx 180 ry 0 rz 180 deg; joints [-138.003, -51.985, -96.255, 46.638, 66.973, -22.499]
  MoveL 5643 to (-35.13, 38.73, 88.06) mm, rotated rx 180 ry 0 rz 180 deg; joints [-138.003, -51.985, -96.255, 46.638, 66.973, -22.499]
  Call Extruder(68.73228)
  MoveL 5644 to (-34.68, 38.4, 88.06) mm, rotated rx 180 ry 0 rz 180 deg; joints [-138.092, -51.992, -96.236, 46.552, 66.929, -22.474]
  MoveL 5645 to (-34.68, 38.4, 88.06) mm, rotated rx 180 ry 0 rz 180 deg; joints [-138.092, -51.992, -96.236, 46.552, 66.929, -22.474]
  Call Extruder(69.06452)
  MoveL 5646 to (-34.22, 38.08, 88.06) mm, rotated rx -180 ry 0 rz -180 deg; joints [-138.182, -51.998, -96.216, 46.466, 66.886, -22.45]
  MoveL 5647 to (-34.22, 38.08, 88.06) mm, rotated rx -180 ry 0 rz -180 deg; joints [-138.182, -51.998, -96.216, 46.466, 66.886, -22.45]
  Call Extruder(69.18223)
  MoveL 5648 to (-34.05, 37.98, 88.06) mm, rotated rx 180 ry 0 rz -180 deg; joints [-138.213, -52.002, -96.205, 46.437, 66.869, -22.443]
  MoveL 5649 to (-34.05, 37.98, 88.06) mm, rotated rx 180 ry 0 rz -180 deg; joints [-138.213, -52.002, -96.205, 46.437, 66.869, -22.443]
  Call Extruder(69.38995)
  MoveL 5650 to (-33.75, 37.8, 88.06) mm, rotated rx 180 ry 0 rz 180 deg; joints [-138.267, -52.008, -96.187, 46.386, 66.84, -22.431]
  MoveL 5651 to (-33.75, 37.8, 88.06) mm, rotated rx 180 ry 0 rz 180 deg; joints [-138.267, -52.008, -96.187, 46.386, 66.84, -22.431]
  Call Extruder(69.59689)
  MoveL 5652 to (-33.45, 37.63, 88.06) mm, rotated rx 180 ry 0 rz -180 deg; joints [-138.322, -52.014, -96.168, 46.335, 66.81, -22.42]
  MoveL 5653 to (-33.45, 37.63, 88.06) mm, rotated rx 180 ry 0 rz -180 deg; joints [-138.322, -52.014, -96.168, 46.335, 66.81, -22.42]
  Call Extruder(69.80305)
  MoveL 5654 to (-33.14, 37.45, 88.06) mm, rotated rx 180 ry 0 rz 180 deg; joints [-138.376, -52.02, -96.149, 46.284, 66.78, -22.408]
  MoveL 5655 to (-33.14, 37.45, 88.06) mm, rotated rx 180 ry 0 rz 180 deg; joints [-138.376, -52.02, -96.149, 46.284, 66.78, -22.408]
  Call Extruder(69.98473)
  MoveL 5656 to (-32.86, 37.31, 88.06) mm, rotated rx 180 ry 0 rz 180 deg; joints [-138.424, -52.026, -96.13, 46.241, 66.753, -22.4]
  MoveL 5657 to (-32.86, 37.31, 88.06) mm, rotated rx 180 ry 0 rz 180 deg; joints [-138.424, -52.026, -96.13, 46.241, 66.753, -22.4]
  Call Extruder(70.14273)
  MoveL 5658 to (-32.62, 37.2, 88.06) mm, rotated rx 180 ry 0 rz -180 deg; joints [-138.464, -52.032, -96.111, 46.204, 66.729, -22.394]
  MoveL 5659 to (-32.62, 37.2, 88.06) mm, rotated rx 180 ry 0 rz -180 deg; joints [-138.464, -52.032, -96.111, 46.204, 66.729, -22.394]
  Call Extruder(70.30013)
  MoveL 5660 to (-32.37, 37.1, 88.06) mm, rotated rx 180 ry 0 rz -180 deg; joints [-138.504, -52.039, -96.091, 46.168, 66.704, -22.389]
  MoveL 5661 to (-32.37, 37.1, 88.06) mm, rotated rx 180 ry 0 rz -180 deg; joints [-138.504, -52.039, -96.091, 46.168, 66.704, -22.389]
  Call Extruder(70.48284)
  MoveL 5662 to (-32.07, 36.98, 88.06) mm, rotated rx 180 ry 0 rz 180 deg; joints [-138.551, -52.046, -96.067, 46.126, 66.676, -22.383]
  MoveL 5663 to (-32.07, 36.98, 88.06) mm, rotated rx 180 ry 0 rz 180 deg; joints [-138.551, -52.046, -96.067, 46.126, 66.676, -22.383]
  Call Extruder(70.66479)
  MoveL 5664 to (-31.78, 36.85, 88.06) mm, rotated rx 180 ry 0 rz -180 deg; joints [-138.597, -52.054, -96.044, 46.084, 66.647, -22.377]
  MoveL 5665 to (-31.78, 36.85, 88.06) mm, rotated rx 180 ry 0 rz -180 deg; joints [-138.597, -52.054, -96.044, 46.084, 66.647, -22.377]
  Call Extruder(70.81212)
  MoveL 5666 to (-31.54, 36.76, 88.06) mm, rotated rx 180 ry 0 rz 180 deg; joints [-138.634, -52.06, -96.023, 46.051, 66.623, -22.373]
  MoveL 5667 to (-31.54, 36.76, 88.06) mm, rotated rx 180 ry 0 rz 180 deg; joints [-138.634, -52.06, -96.023, 46.051, 66.623, -22.373]
  Call Extruder(70.92536)
  MoveL 5668 to (-31.35, 36.7, 88.06) mm, rotated rx 180 ry 0 rz -180 deg; joints [-138.662, -52.066, -96.006, 46.027, 66.605, -22.371]
  MoveL 5669 to (-31.35, 36.7, 88.06) mm, rotated rx 180 ry 0 rz -180 deg; joints [-138.662, -52.066, -96.006, 46.027, 66.605, -22.371]
  Call Extruder(71.03815)
  MoveL 5670 to (-31.17, 36.64, 88.06) mm, rotated rx 180 ry 0 rz 180 deg; joints [-138.69, -52.072, -95.989, 46.002, 66.586, -22.368]
  MoveL 5671 to (-31.17, 36.64, 88.06) mm, rotated rx 180 ry 0 rz 180 deg; joints [-138.69, -52.072, -95.989, 46.002, 66.586, -22.368]
  Call Extruder(71.15050)
  MoveL 5672 to (-30.98, 36.58, 88.06) mm, rotated rx 180 ry 0 rz 180 deg; joints [-138.718, -52.077, -95.972, 45.978, 66.567, -22.366]
  MoveL 5673 to (-30.98, 36.58, 88.06) mm, rotated rx 180 ry 0 rz 180 deg; joints [-138.718, -52.077, -95.972, 45.978, 66.567, -22.366]
  Call Extruder(71.26240)
  MoveL 5674 to (-30.79, 36.52, 88.06) mm, rotated rx 180 ry 0 rz 180 deg; joints [-138.745, -52.083, -95.955, 45.954, 66.549, -22.364]
  MoveL 5675 to (-30.79, 36.52, 88.06) mm, rotated rx 180 ry 0 rz 180 deg; joints [-138.745, -52.083, -95.955, 45.954, 66.549, -22.364]
  Call Extruder(71.38380)
  MoveL 5676 to (-30.58, 36.45, 88.06) mm, rotated rx 180 ry 0 rz 180 deg; joints [-138.776, -52.089, -95.936, 45.927, 66.528, -22.362]
  MoveL 5677 to (-30.58, 36.45, 88.06) mm, rotated rx 180 ry 0 rz 180 deg; joints [-138.776, -52.089, -95.936, 45.927, 66.528, -22.362]
  Call Extruder(71.51459)
  MoveL 5678 to (-30.36, 36.39, 88.06) mm, rotated rx 180 ry 0 rz 180 deg; joints [-138.808, -52.096, -95.915, 45.899, 66.506, -22.361]
  MoveL 5679 to (-30.36, 36.39, 88.06) mm, rotated rx 180 ry 0 rz 180 deg; joints [-138.808, -52.096, -95.915, 45.899, 66.506, -22.361]
  Call Extruder(71.64482)
  MoveL 5680 to (-30.14, 36.32, 88.06) mm, rotated rx 180 ry 0 rz 180 deg; joints [-138.84, -52.102, -95.894, 45.871, 66.484, -22.359]
  MoveL 5681 to (-30.14, 36.32, 88.06) mm, rotated rx 180 ry 0 rz 180 deg; joints [-138.84, -52.102, -95.894, 45.871, 66.484, -22.359]
  Call Extruder(71.77448)
  MoveL 5682 to (-29.91, 36.25, 88.06) mm, rotated rx -180 ry 0 rz -180 deg; joints [-138.873, -52.109, -95.872, 45.843, 66.462, -22.357]
  MoveL 5683 to (-29.91, 36.25, 88.06) mm, rotated rx -180 ry 0 rz -180 deg; joints [-138.873, -52.109, -95.872, 45.843, 66.462, -22.357]
  Call Extruder(71.90358)
  MoveL 5684 to (-29.69, 36.18, 88.06) mm, rotated rx 180 ry 0 rz -180 deg; joints [-138.905, -52.116, -95.851, 45.815, 66.439, -22.355]
  MoveL 5685 to (-29.69, 36.18, 88.06) mm, rotated rx 180 ry 0 rz -180 deg; joints [-138.905, -52.116, -95.851, 45.815, 66.439, -22.355]
  Call Extruder(72.01865)
  MoveL 5686 to (-29.48, 36.14, 88.06) mm, rotated rx 180 ry 0 rz 180 deg; joints [-138.932, -52.123, -95.83, 45.792, 66.419, -22.355]
  MoveL 5687 to (-29.48, 36.14, 88.06) mm, rotated rx 180 ry 0 rz 180 deg; joints [-138.932, -52.123, -95.83, 45.792, 66.419, -22.355]
  Call Extruder(72.13327)
  MoveL 5688 to (-29.28, 36.09, 88.06) mm, rotated rx -180 ry 0 rz 180 deg; joints [-138.96, -52.13, -95.809, 45.768, 66.399, -22.355]
  MoveL 5689 to (-29.28, 36.09, 88.06) mm, rotated rx -180 ry 0 rz 180 deg; joints [-138.96, -52.13, -95.809, 45.768, 66.399, -22.355]
  Call Extruder(72.24744)
  MoveL 5690 to (-29.08, 36.05, 88.06) mm, rotated rx 180 ry 0 rz -180 deg; joints [-138.987, -52.137, -95.788, 45.746, 66.378, -22.356]
  MoveL 5691 to (-29.08, 36.05, 88.06) mm, rotated rx 180 ry 0 rz -180 deg; joints [-138.987, -52.137, -95.788, 45.746, 66.378, -22.356]
  Call Extruder(72.36115)
  MoveL 5692 to (-28.87, 36, 88.06) mm, rotated rx 180 ry 0 rz 180 deg; joints [-139.014, -52.144, -95.766, 45.722, 66.358, -22.356]
  MoveL 5693 to (-28.87, 36, 88.06) mm, rotated rx 180 ry 0 rz 180 deg; joints [-139.014, -52.144, -95.766, 45.722, 66.358, -22.356]
  Call Extruder(72.48657)
  MoveL 5694 to (-28.64, 35.96, 88.06) mm, rotated rx -180 ry 0 rz 180 deg; joints [-139.044, -52.152, -95.743, 45.697, 66.335, -22.356]
  MoveL 5695 to (-28.64, 35.96, 88.06) mm, rotated rx -180 ry 0 rz 180 deg; joints [-139.044, -52.152, -95.743, 45.697, 66.335, -22.356]
  Call Extruder(72.62355)
  MoveL 5696 to (-28.4, 35.91, 88.06) mm, rotated rx -180 ry 0 rz -180 deg; joints [-139.077, -52.16, -95.716, 45.67, 66.31, -22.357]
  MoveL 5697 to (-28.4, 35.91, 88.06) mm, rotated rx -180 ry 0 rz -180 deg; joints [-139.077, -52.16, -95.716, 45.67, 66.31, -22.357]
  Call Extruder(72.75992)
  MoveL 5698 to (-28.15, 35.86, 88.06) mm, rotated rx -180 ry 0 rz 180 deg; joints [-139.109, -52.169, -95.69, 45.643, 66.285, -22.358]
  MoveL 5699 to (-28.15, 35.86, 88.06) mm, rotated rx -180 ry 0 rz 180 deg; joints [-139.109, -52.169, -95.69, 45.643, 66.285, -22.358]
  Call Extruder(72.89567)
  MoveL 5700 to (-27.9, 35.81, 88.06) mm, rotated rx 180 ry 0 rz 180 deg; joints [-139.142, -52.177, -95.663, 45.615, 66.26, -22.358]
  MoveL 5701 to (-27.9, 35.81, 88.06) mm, rotated rx 180 ry 0 rz 180 deg; joints [-139.142, -52.177, -95.663, 45.615, 66.26, -22.358]
  Call Extruder(73.03082)
  MoveL 5702 to (-27.65, 35.76, 88.06) mm, rotated rx 180 ry 0 rz -180 deg; joints [-139.174, -52.186, -95.636, 45.588, 66.236, -22.359]
  MoveL 5703 to (-27.65, 35.76, 88.06) mm, rotated rx 180 ry 0 rz -180 deg; joints [-139.174, -52.186, -95.636, 45.588, 66.236, -22.359]
  Call Extruder(73.16536)
  MoveL 5704 to (-27.4, 35.71, 88.06) mm, rotated rx 180 ry 0 rz 180 deg; joints [-139.207, -52.195, -95.61, 45.561, 66.211, -22.36]
  MoveL 5705 to (-27.4, 35.71, 88.06) mm, rotated rx 180 ry 0 rz 180 deg; joints [-139.207, -52.195, -95.61, 45.561, 66.211, -22.36]
  Call Extruder(73.29928)
  MoveL 5706 to (-27.15, 35.66, 88.06) mm, rotated rx 180 ry 0 rz 180 deg; joints [-139.239, -52.204, -95.583, 45.534, 66.186, -22.361]
  MoveL 5707 to (-27.15, 35.66, 88.06) mm, rotated rx 180 ry 0 rz 180 deg; joints [-139.239, -52.204, -95.583, 45.534, 66.186, -22.361]
  Call Extruder(73.44714)
  MoveL 5708 to (-26.87, 35.61, 88.06) mm, rotated rx -180 ry 0 rz -180 deg; joints [-139.275, -52.213, -95.553, 45.504, 66.158, -22.362]
  MoveL 5709 to (-26.87, 35.61, 88.06) mm, rotated rx -180 ry 0 rz -180 deg; joints [-139.275, -52.213, -95.553, 45.504, 66.158, -22.362]
  Call Extruder(73.60888)
  MoveL 5710 to (-26.57, 35.56, 88.06) mm, rotated rx -180 ry 0 rz 180 deg; joints [-139.313, -52.225, -95.519, 45.473, 66.127, -22.364]
  MoveL 5711 to (-26.57, 35.56, 88.06) mm, rotated rx -180 ry 0 rz 180 deg; joints [-139.313, -52.225, -95.519, 45.473, 66.127, -22.364]
  Call Extruder(73.76989)
  MoveL 5712 to (-26.26, 35.51, 88.06) mm, rotated rx -180 ry 0 rz -180 deg; joints [-139.351, -52.236, -95.484, 45.441, 66.097, -22.367]
  MoveL 5713 to (-26.26, 35.51, 88.06) mm, rotated rx -180 ry 0 rz -180 deg; joints [-139.351, -52.236, -95.484, 45.441, 66.097, -22.367]
  Call Extruder(73.93017)
  MoveL 5714 to (-25.96, 35.46, 88.06) mm, rotated rx -180 ry 0 rz 180 deg; joints [-139.39, -52.247, -95.45, 45.41, 66.066, -22.369]
  MoveL 5715 to (-25.96, 35.46, 88.06) mm, rotated rx -180 ry 0 rz 180 deg; joints [-139.39, -52.247, -95.45, 45.41, 66.066, -22.369]
  Call Extruder(74.08972)
  MoveL 5716 to (-25.65, 35.42, 88.06) mm, rotated rx 180 ry 0 rz 180 deg; joints [-139.428, -52.258, -95.416, 45.379, 66.035, -22.371]
  MoveL 5717 to (-25.65, 35.42, 88.06) mm, rotated rx 180 ry 0 rz 180 deg; joints [-139.428, -52.258, -95.416, 45.379, 66.035, -22.371]
  Call Extruder(74.24855)
  MoveL 5718 to (-25.34, 35.37, 88.06) mm, rotated rx 180 ry 0 rz -180 deg; joints [-139.466, -52.269, -95.382, 45.347, 66.004, -22.373]
  MoveL 5719 to (-25.34, 35.37, 88.06) mm, rotated rx 180 ry 0 rz -180 deg; joints [-139.466, -52.269, -95.382, 45.347, 66.004, -22.373]
  Call Extruder(74.42721)
  MoveL 5720 to (-25, 35.32, 88.06) mm, rotated rx -180 ry 0 rz -180 deg; joints [-139.508, -52.282, -95.342, 45.313, 65.97, -22.377]
  MoveL 5721 to (-25, 35.32, 88.06) mm, rotated rx -180 ry 0 rz -180 deg; joints [-139.508, -52.282, -95.342, 45.313, 65.97, -22.377]
  Call Extruder(74.62566)
  MoveL 5722 to (-24.61, 35.27, 88.06) mm, rotated rx 180 ry 0 rz 180 deg; joints [-139.554, -52.297, -95.297, 45.276, 65.931, -22.381]
  MoveL 5723 to (-24.61, 35.27, 88.06) mm, rotated rx 180 ry 0 rz 180 deg; joints [-139.554, -52.297, -95.297, 45.276, 65.931, -22.381]
  Call Extruder(74.82323)
  MoveL 5724 to (-24.22, 35.23, 88.06) mm, rotated rx 180 ry 0 rz 180 deg; joints [-139.6, -52.312, -95.252, 45.239, 65.892, -22.386]
  MoveL 5725 to (-24.22, 35.23, 88.06) mm, rotated rx 180 ry 0 rz 180 deg; joints [-139.6, -52.312, -95.252, 45.239, 65.892, -22.386]
  Call Extruder(75.01994)
  MoveL 5726 to (-23.83, 35.18, 88.06) mm, rotated rx -180 ry 0 rz 180 deg; joints [-139.647, -52.327, -95.206, 45.202, 65.853, -22.391]
  MoveL 5727 to (-23.83, 35.18, 88.06) mm, rotated rx -180 ry 0 rz 180 deg; joints [-139.647, -52.327, -95.206, 45.202, 65.853, -22.391]
  Call Extruder(75.21578)
  MoveL 5728 to (-23.45, 35.14, 88.06) mm, rotated rx -180 ry 0 rz 180 deg; joints [-139.693, -52.342, -95.161, 45.165, 65.814, -22.395]
  MoveL 5729 to (-23.45, 35.14, 88.06) mm, rotated rx -180 ry 0 rz 180 deg; joints [-139.693, -52.342, -95.161, 45.165, 65.814, -22.395]
  Call Extruder(75.51117)
  MoveL 5730 to (-22.86, 35.09, 88.06) mm, rotated rx 180 ry 0 rz 180 deg; joints [-139.76, -52.366, -95.089, 45.112, 65.754, -22.405]
  MoveL 5731 to (-22.86, 35.09, 88.06) mm, rotated rx 180 ry 0 rz 180 deg; joints [-139.76, -52.366, -95.089, 45.112, 65.754, -22.405]
  Call Extruder(75.80523)
  MoveL 5732 to (-22.27, 35.04, 88.06) mm, rotated rx -180 ry 0 rz 180 deg; joints [-139.826, -52.389, -95.017, 45.06, 65.694, -22.414]
  MoveL 5733 to (-22.27, 35.04, 88.06) mm, rotated rx -180 ry 0 rz 180 deg; joints [-139.826, -52.389, -95.017, 45.06, 65.694, -22.414]
  Call Extruder(76.09796)
  MoveL 5734 to (-21.68, 35, 88.06) mm, rotated rx 180 ry 0 rz 180 deg; joints [-139.893, -52.413, -94.945, 45.007, 65.635, -22.424]
  MoveL 5735 to (-21.68, 35, 88.06) mm, rotated rx 180 ry 0 rz 180 deg; joints [-139.893, -52.413, -94.945, 45.007, 65.635, -22.424]
  Call Extruder(76.67141)
  MoveL 5736 to (-20.52, 34.95, 88.06) mm, rotated rx 180 ry 0 rz -180 deg; joints [-140.019, -52.462, -94.797, 44.912, 65.517, -22.448]
  MoveL 5737 to (-20.52, 34.95, 88.06) mm, rotated rx 180 ry 0 rz -180 deg; joints [-140.019, -52.462, -94.797, 44.912, 65.517, -22.448]
  Call Extruder(77.38537)
  MoveL 5738 to (-19.06, 34.91, 88.06) mm, rotated rx 180 ry 0 rz 180 deg; joints [-140.173, -52.524, -94.61, 44.795, 65.37, -22.48]
  Call Extruder(194.23211)
  MoveL 5739 to (219.06, 34.91, 88.06) mm, rotated rx -180 ry 0 rz 180 deg; joints [-155.896, -69.983, -52.2, 40.03, 39.416, -32.981]
  Call Extruder(194.66067)
  MoveL 5740 to (219.94, 34.93, 88.06) mm, rotated rx -180 ry 0 rz 180 deg; joints [-155.931, -70.082, -51.985, 40.075, 39.308, -33.063]
  MoveL 5741 to (219.94, 34.93, 88.06) mm, rotated rx -180 ry 0 rz 180 deg; joints [-155.931, -70.082, -51.985, 40.075, 39.308, -33.063]
  Call Extruder(195.23412)
  MoveL 5742 to (221.1, 34.97, 88.06) mm, rotated rx 180 ry 0 rz 180 deg; joints [-155.975, -70.216, -51.695, 40.14, 39.165, -33.177]
  MoveL 5743 to (221.1, 34.97, 88.06) mm, rotated rx 180 ry 0 rz 180 deg; joints [-155.975, -70.216, -51.695, 40.14, 39.165, -33.177]
  Call Extruder(195.66843)
  MoveL 5744 to (221.97, 35.02, 88.06) mm, rotated rx -180 ry 0 rz -180 deg; joints [-156.007, -70.318, -51.475, 40.191, 39.057, -33.265]
  MoveL 5745 to (221.97, 35.02, 88.06) mm, rotated rx -180 ry 0 rz -180 deg; joints [-156.007, -70.318, -51.475, 40.191, 39.057, -33.265]
  Call Extruder(195.96249)
  MoveL 5746 to (222.56, 35.07, 88.06) mm, rotated rx 180 ry 0 rz 180 deg; joints [-156.027, -70.388, -51.324, 40.229, 38.985, -33.327]
  MoveL 5747 to (222.56, 35.07, 88.06) mm, rotated rx 180 ry 0 rz 180 deg; joints [-156.027, -70.388, -51.324, 40.229, 38.985, -33.327]
  Call Extruder(196.25788)
  MoveL 5748 to (223.15, 35.11, 88.06) mm, rotated rx 180 ry 0 rz 180 deg; joints [-156.047, -70.458, -51.173, 40.267, 38.912, -33.39]
  MoveL 5749 to (223.15, 35.11, 88.06) mm, rotated rx 180 ry 0 rz 180 deg; joints [-156.047, -70.458, -51.173, 40.267, 38.912, -33.39]
  Call Extruder(196.50411)
  MoveL 5750 to (223.64, 35.16, 88.06) mm, rotated rx 180 ry 0 rz 180 deg; joints [-156.062, -70.516, -51.047, 40.3, 38.852, -33.443]
  MoveL 5751 to (223.64, 35.16, 88.06) mm, rotated rx 180 ry 0 rz 180 deg; joints [-156.062, -70.516, -51.047, 40.3, 38.852, -33.443]
  Call Extruder(196.70082)
  MoveL 5752 to (224.03, 35.21, 88.06) mm, rotated rx 180 ry 0 rz 180 deg; joints [-156.074, -70.563, -50.946, 40.329, 38.804, -33.487]
  MoveL 5753 to (224.03, 35.21, 88.06) mm, rotated rx 180 ry 0 rz 180 deg; joints [-156.074, -70.563, -50.946, 40.329, 38.804, -33.487]
  Call Extruder(196.89840)
  MoveL 5754 to (224.42, 35.25, 88.06) mm, rotated rx 180 ry 0 rz 180 deg; joints [-156.086, -70.61, -50.845, 40.357, 38.756, -33.531]
  MoveL 5755 to (224.42, 35.25, 88.06) mm, rotated rx 180 ry 0 rz 180 deg; joints [-156.086, -70.61, -50.845, 40.357, 38.756, -33.531]
  Call Extruder(197.09684)
  MoveL 5756 to (224.8, 35.3, 88.06) mm, rotated rx -180 ry 0 rz 180 deg; joints [-156.097, -70.658, -50.743, 40.385, 38.708, -33.575]
  MoveL 5757 to (224.8, 35.3, 88.06) mm, rotated rx -180 ry 0 rz 180 deg; joints [-156.097, -70.658, -50.743, 40.385, 38.708, -33.575]
  Call Extruder(197.29615)
  MoveL 5758 to (225.19, 35.34, 88.06) mm, rotated rx 180 ry 0 rz 180 deg; joints [-156.109, -70.705, -50.642, 40.414, 38.661, -33.62]
  MoveL 5759 to (225.19, 35.34, 88.06) mm, rotated rx 180 ry 0 rz 180 deg; joints [-156.109, -70.705, -50.642, 40.414, 38.661, -33.62]
  Call Extruder(197.45497)
  MoveL 5760 to (225.5, 35.39, 88.06) mm, rotated rx 180 ry 0 rz 180 deg; joints [-156.117, -70.743, -50.56, 40.439, 38.623, -33.657]
  MoveL 5761 to (225.5, 35.39, 88.06) mm, rotated rx 180 ry 0 rz 180 deg; joints [-156.117, -70.743, -50.56, 40.439, 38.623, -33.657]
  Call Extruder(197.61452)
  MoveL 5762 to (225.8, 35.44, 88.06) mm, rotated rx 180 ry 0 rz 180 deg; joints [-156.125, -70.781, -50.478, 40.464, 38.585, -33.694]
  MoveL 5763 to (225.8, 35.44, 88.06) mm, rotated rx 180 ry 0 rz 180 deg; joints [-156.125, -70.781, -50.478, 40.464, 38.585, -33.694]
  Call Extruder(197.77480)
  MoveL 5764 to (226.11, 35.49, 88.06) mm, rotated rx 180 ry 0 rz 180 deg; joints [-156.133, -70.819, -50.396, 40.489, 38.547, -33.731]
  MoveL 5765 to (226.11, 35.49, 88.06) mm, rotated rx 180 ry 0 rz 180 deg; joints [-156.133, -70.819, -50.396, 40.489, 38.547, -33.731]
  Call Extruder(197.93580)
  MoveL 5766 to (226.41, 35.54, 88.06) mm, rotated rx -180 ry 0 rz -180 deg; joints [-156.141, -70.857, -50.314, 40.514, 38.51, -33.768]
  MoveL 5767 to (226.41, 35.54, 88.06) mm, rotated rx -180 ry 0 rz -180 deg; joints [-156.141, -70.857, -50.314, 40.514, 38.51, -33.768]
  Call Extruder(198.09753)
  MoveL 5768 to (226.72, 35.59, 88.06) mm, rotated rx 180 ry 0 rz -180 deg; joints [-156.149, -70.895, -50.232, 40.539, 38.472, -33.806]
  MoveL 5769 to (226.72, 35.59, 88.06) mm, rotated rx 180 ry 0 rz -180 deg; joints [-156.149, -70.895, -50.232, 40.539, 38.472, -33.806]
  Call Extruder(198.25999)
  MoveL 5770 to (227.03, 35.63, 88.06) mm, rotated rx -180 ry 0 rz 180 deg; joints [-156.157, -70.933, -50.15, 40.564, 38.434, -33.844]
  MoveL 5771 to (227.03, 35.63, 88.06) mm, rotated rx -180 ry 0 rz 180 deg; joints [-156.157, -70.933, -50.15, 40.564, 38.434, -33.844]
  Call Extruder(198.39392)
  MoveL 5772 to (227.27, 35.68, 88.06) mm, rotated rx 180 ry 0 rz 180 deg; joints [-156.162, -70.965, -50.082, 40.587, 38.403, -33.876]
  MoveL 5773 to (227.27, 35.68, 88.06) mm, rotated rx 180 ry 0 rz 180 deg; joints [-156.162, -70.965, -50.082, 40.587, 38.403, -33.876]
  Call Extruder(198.52846)
  MoveL 5774 to (227.52, 35.73, 88.06) mm, rotated rx 180 ry 0 rz 180 deg; joints [-156.168, -70.997, -50.014, 40.609, 38.372, -33.908]
  MoveL 5775 to (227.52, 35.73, 88.06) mm, rotated rx 180 ry 0 rz 180 deg; joints [-156.168, -70.997, -50.014, 40.609, 38.372, -33.908]
  Call Extruder(198.66360)
  MoveL 5776 to (227.77, 35.78, 88.06) mm, rotated rx -180 ry 0 rz 180 deg; joints [-156.173, -71.029, -49.945, 40.632, 38.342, -33.941]
  MoveL 5777 to (227.77, 35.78, 88.06) mm, rotated rx -180 ry 0 rz 180 deg; joints [-156.173, -71.029, -49.945, 40.632, 38.342, -33.941]
  Call Extruder(198.79936)
  MoveL 5778 to (228.02, 35.83, 88.06) mm, rotated rx -180 ry 0 rz 180 deg; joints [-156.179, -71.061, -49.877, 40.655, 38.311, -33.973]
  MoveL 5779 to (228.02, 35.83, 88.06) mm, rotated rx -180 ry 0 rz 180 deg; joints [-156.179, -71.061, -49.877, 40.655, 38.311, -33.973]
  Call Extruder(198.93573)
  MoveL 5780 to (228.27, 35.88, 88.06) mm, rotated rx 180 ry 0 rz -180 deg; joints [-156.185, -71.093, -49.808, 40.677, 38.28, -34.006]
  MoveL 5781 to (228.27, 35.88, 88.06) mm, rotated rx 180 ry 0 rz -180 deg; joints [-156.185, -71.093, -49.808, 40.677, 38.28, -34.006]
  Call Extruder(199.07271)
  MoveL 5782 to (228.52, 35.93, 88.06) mm, rotated rx 180 ry 0 rz 180 deg; joints [-156.19, -71.124, -49.74, 40.7, 38.249, -34.039]
  MoveL 5783 to (228.52, 35.93, 88.06) mm, rotated rx 180 ry 0 rz 180 deg; joints [-156.19, -71.124, -49.74, 40.7, 38.249, -34.039]
  Call Extruder(199.21030)
  MoveL 5784 to (228.77, 35.98, 88.06) mm, rotated rx 180 ry 0 rz 180 deg; joints [-156.196, -71.156, -49.671, 40.723, 38.218, -34.071]
  MoveL 5785 to (228.77, 35.98, 88.06) mm, rotated rx 180 ry 0 rz 180 deg; joints [-156.196, -71.156, -49.671, 40.723, 38.218, -34.071]
  Call Extruder(199.32402)
  MoveL 5786 to (228.97, 36.03, 88.06) mm, rotated rx 180 ry 0 rz 180 deg; joints [-156.2, -71.183, -49.615, 40.742, 38.193, -34.099]
  MoveL 5787 to (228.97, 36.03, 88.06) mm, rotated rx 180 ry 0 rz 180 deg; joints [-156.2, -71.183, -49.615, 40.742, 38.193, -34.099]
  Call Extruder(199.43819)
  MoveL 5788 to (229.18, 36.07, 88.06) mm, rotated rx 180 ry 0 rz 180 deg; joints [-156.204, -71.209, -49.558, 40.762, 38.168, -34.127]
  MoveL 5789 to (229.18, 36.07, 88.06) mm, rotated rx 180 ry 0 rz 180 deg; joints [-156.204, -71.209, -49.558, 40.762, 38.168, -34.127]
  Call Extruder(199.55281)
  MoveL 5790 to (229.38, 36.12, 88.06) mm, rotated rx 180 ry 0 rz 180 deg; joints [-156.208, -71.236, -49.501, 40.782, 38.142, -34.154]
  MoveL 5791 to (229.38, 36.12, 88.06) mm, rotated rx 180 ry 0 rz 180 deg; joints [-156.208, -71.236, -49.501, 40.782, 38.142, -34.154]
  Call Extruder(199.66788)
  MoveL 5792 to (229.59, 36.16, 88.06) mm, rotated rx 180 ry 0 rz -180 deg; joints [-156.212, -71.262, -49.444, 40.801, 38.117, -34.182]
  MoveL 5793 to (229.59, 36.16, 88.06) mm, rotated rx 180 ry 0 rz -180 deg; joints [-156.212, -71.262, -49.444, 40.801, 38.117, -34.182]
  Call Extruder(199.79012)
  MoveL 5794 to (229.8, 36.22, 88.06) mm, rotated rx 180 ry 0 rz 180 deg; joints [-156.216, -71.291, -49.384, 40.824, 38.091, -34.212]
  MoveL 5795 to (229.8, 36.22, 88.06) mm, rotated rx 180 ry 0 rz 180 deg; joints [-156.216, -71.291, -49.384, 40.824, 38.091, -34.212]
  Call Extruder(199.91978)
  MoveL 5796 to (230.02, 36.28, 88.06) mm, rotated rx 180 ry 0 rz -180 deg; joints [-156.219, -71.321, -49.319, 40.849, 38.063, -34.246]
  MoveL 5797 to (230.02, 36.28, 88.06) mm, rotated rx 180 ry 0 rz -180 deg; joints [-156.219, -71.321, -49.319, 40.849, 38.063, -34.246]
  Call Extruder(200.05001)
  MoveL 5798 to (230.25, 36.35, 88.06) mm, rotated rx -180 ry 0 rz 180 deg; joints [-156.221, -71.351, -49.255, 40.874, 38.035, -34.28]
  MoveL 5799 to (230.25, 36.35, 88.06) mm, rotated rx -180 ry 0 rz 180 deg; joints [-156.221, -71.351, -49.255, 40.874, 38.035, -34.28]
  Call Extruder(200.18081)
  MoveL 5800 to (230.47, 36.42, 88.06) mm, rotated rx 180 ry 0 rz -180 deg; joints [-156.224, -71.381, -49.19, 40.899, 38.008, -34.313]
  MoveL 5801 to (230.47, 36.42, 88.06) mm, rotated rx 180 ry 0 rz -180 deg; joints [-156.224, -71.381, -49.19, 40.899, 38.008, -34.313]
  Call Extruder(200.31217)
  MoveL 5802 to (230.7, 36.49, 88.06) mm, rotated rx 180 ry 0 rz 180 deg; joints [-156.227, -71.411, -49.125, 40.924, 37.98, -34.347]
  MoveL 5803 to (230.7, 36.49, 88.06) mm, rotated rx 180 ry 0 rz 180 deg; joints [-156.227, -71.411, -49.125, 40.924, 37.98, -34.347]
  Call Extruder(200.40859)
  MoveL 5804 to (230.86, 36.54, 88.06) mm, rotated rx 180 ry 0 rz -180 deg; joints [-156.229, -71.433, -49.078, 40.943, 37.96, -34.372]
  MoveL 5805 to (230.86, 36.54, 88.06) mm, rotated rx 180 ry 0 rz -180 deg; joints [-156.229, -71.433, -49.078, 40.943, 37.96, -34.372]
  Call Extruder(200.52476)
  MoveL 5806 to (231.05, 36.6, 88.06) mm, rotated rx -180 ry 0 rz 180 deg; joints [-156.231, -71.46, -49.021, 40.965, 37.936, -34.402]
  MoveL 5807 to (231.05, 36.6, 88.06) mm, rotated rx -180 ry 0 rz 180 deg; joints [-156.231, -71.46, -49.021, 40.965, 37.936, -34.402]
  Call Extruder(200.64140)
  MoveL 5808 to (231.25, 36.67, 88.06) mm, rotated rx 180 ry 0 rz 180 deg; joints [-156.233, -71.487, -48.964, 40.988, 37.912, -34.432]
  MoveL 5809 to (231.25, 36.67, 88.06) mm, rotated rx 180 ry 0 rz 180 deg; joints [-156.233, -71.487, -48.964, 40.988, 37.912, -34.432]
  Call Extruder(200.75852)
  MoveL 5810 to (231.44, 36.73, 88.06) mm, rotated rx -180 ry 0 rz -180 deg; joints [-156.235, -71.513, -48.907, 41.011, 37.888, -34.463]
  MoveL 5811 to (231.44, 36.73, 88.06) mm, rotated rx -180 ry 0 rz -180 deg; joints [-156.235, -71.513, -48.907, 41.011, 37.888, -34.463]
  Call Extruder(200.87612)
  MoveL 5812 to (231.64, 36.79, 88.06) mm, rotated rx 180 ry 0 rz 180 deg; joints [-156.237, -71.54, -48.85, 41.034, 37.864, -34.493]
  MoveL 5813 to (231.64, 36.79, 88.06) mm, rotated rx 180 ry 0 rz 180 deg; joints [-156.237, -71.54, -48.85, 41.034, 37.864, -34.493]
  Call Extruder(201.05807)
  MoveL 5814 to (231.93, 36.91, 88.06) mm, rotated rx 180 ry 0 rz 180 deg; joints [-156.238, -71.582, -48.761, 41.073, 37.828, -34.543]
  MoveL 5815 to (231.93, 36.91, 88.06) mm, rotated rx 180 ry 0 rz 180 deg; joints [-156.238, -71.582, -48.761, 41.073, 37.828, -34.543]
  Call Extruder(201.24079)
  MoveL 5816 to (232.22, 37.03, 88.06) mm, rotated rx 180 ry 0 rz 180 deg; joints [-156.238, -71.623, -48.672, 41.112, 37.792, -34.593]
  MoveL 5817 to (232.22, 37.03, 88.06) mm, rotated rx 180 ry 0 rz 180 deg; joints [-156.238, -71.623, -48.672, 41.112, 37.792, -34.593]
  Call Extruder(201.41121)
  MoveL 5818 to (232.49, 37.15, 88.06) mm, rotated rx -180 ry 0 rz 180 deg; joints [-156.239, -71.662, -48.59, 41.149, 37.758, -34.639]
  MoveL 5819 to (232.49, 37.15, 88.06) mm, rotated rx -180 ry 0 rz 180 deg; joints [-156.239, -71.662, -48.59, 41.149, 37.758, -34.639]
  Call Extruder(201.56921)
  MoveL 5820 to (232.74, 37.26, 88.06) mm, rotated rx 180 ry 0 rz 180 deg; joints [-156.239, -71.697, -48.514, 41.183, 37.728, -34.683]
  MoveL 5821 to (232.74, 37.26, 88.06) mm, rotated rx 180 ry 0 rz 180 deg; joints [-156.239, -71.697, -48.514, 41.183, 37.728, -34.683]
  Call Extruder(201.72781)
  MoveL 5822 to (232.99, 37.36, 88.06) mm, rotated rx -180 ry 0 rz -180 deg; joints [-156.239, -71.733, -48.437, 41.217, 37.697, -34.726]
  MoveL 5823 to (232.99, 37.36, 88.06) mm, rotated rx -180 ry 0 rz -180 deg; joints [-156.239, -71.733, -48.437, 41.217, 37.697, -34.726]
  Call Extruder(201.93398)
  MoveL 5824 to (233.29, 37.54, 88.06) mm, rotated rx -180 ry 0 rz 180 deg; joints [-156.236, -71.779, -48.339, 41.267, 37.66, -34.787]
  MoveL 5825 to (233.29, 37.54, 88.06) mm, rotated rx -180 ry 0 rz 180 deg; joints [-156.236, -71.779, -48.339, 41.267, 37.66, -34.787]
  Call Extruder(202.14092)
  MoveL 5826 to (233.6, 37.71, 88.06) mm, rotated rx 180 ry 0 rz 180 deg; joints [-156.232, -71.825, -48.24, 41.317, 37.622, -34.848]
  MoveL 5827 to (233.6, 37.71, 88.06) mm, rotated rx 180 ry 0 rz 180 deg; joints [-156.232, -71.825, -48.24, 41.317, 37.622, -34.848]
  Call Extruder(202.34865)
  MoveL 5828 to (233.9, 37.89, 88.06) mm, rotated rx 180 ry 0 rz 180 deg; joints [-156.228, -71.872, -48.141, 41.367, 37.585, -34.908]
  MoveL 5829 to (233.9, 37.89, 88.06) mm, rotated rx 180 ry 0 rz 180 deg; joints [-156.228, -71.872, -48.141, 41.367, 37.585, -34.908]
  Call Extruder(202.55715)
  MoveL 5830 to (234.21, 38.06, 88.06) mm, rotated rx 180 ry 0 rz 180 deg; joints [-156.224, -71.918, -48.042, 41.417, 37.548, -34.97]
  MoveL 5831 to (234.21, 38.06, 88.06) mm, rotated rx 180 ry 0 rz 180 deg; joints [-156.224, -71.918, -48.042, 41.417, 37.548, -34.97]
  Call Extruder(202.73669)
  MoveL 5832 to (234.45, 38.24, 88.06) mm, rotated rx 180 ry 0 rz 180 deg; joints [-156.218, -71.957, -47.958, 41.464, 37.518, -35.024]
  MoveL 5833 to (234.45, 38.24, 88.06) mm, rotated rx 180 ry 0 rz 180 deg; joints [-156.218, -71.957, -47.958, 41.464, 37.518, -35.024]
  Call Extruder(203.07011)
  MoveL 5834 to (234.9, 38.57, 88.06) mm, rotated rx 180 ry 0 rz 180 deg; joints [-156.206, -72.03, -47.803, 41.551, 37.463, -35.127]
  MoveL 5835 to (234.9, 38.57, 88.06) mm, rotated rx 180 ry 0 rz 180 deg; joints [-156.206, -72.03, -47.803, 41.551, 37.463, -35.127]
  Call Extruder(203.40471)
  MoveL 5836 to (235.35, 38.9, 88.06) mm, rotated rx -180 ry 0 rz 180 deg; joints [-156.195, -72.103, -47.648, 41.638, 37.408, -35.229]
  Call Extruder(204.23266)
  MoveL 5837 to (236.39, 39.81, 88.06) mm, rotated rx -180 ry 0 rz 180 deg; joints [-156.154, -72.28, -47.271, 41.868, 37.283, -35.493]
  Call Extruder(205.06060)
  MoveL 5838 to (237.3, 40.85, 88.06) mm, rotated rx -180 ry 0 rz 180 deg; joints [-156.097, -72.449, -46.91, 42.113, 37.174, -35.765]
  Call Extruder(205.22791)
  MoveL 5839 to (237.47, 41.07, 88.06) mm, rotated rx 180 ry 0 rz 180 deg; joints [-156.083, -72.482, -46.84, 42.164, 37.154, -35.821]
  MoveL 5840 to (237.47, 41.07, 88.06) mm, rotated rx 180 ry 0 rz 180 deg; joints [-156.083, -72.482, -46.84, 42.164, 37.154, -35.821]
  Call Extruder(205.56133)
  MoveL 5841 to (237.79, 41.52, 88.06) mm, rotated rx -180 ry 0 rz 180 deg; joints [-156.055, -72.548, -46.701, 42.267, 37.116, -35.933]
  MoveL 5842 to (237.79, 41.52, 88.06) mm, rotated rx -180 ry 0 rz 180 deg; joints [-156.055, -72.548, -46.701, 42.267, 37.116, -35.933]
  Call Extruder(205.89358)
  MoveL 5843 to (238.12, 41.98, 88.06) mm, rotated rx 180 ry 0 rz -180 deg; joints [-156.028, -72.614, -46.56, 42.37, 37.077, -36.045]
  MoveL 5844 to (238.12, 41.98, 88.06) mm, rotated rx 180 ry 0 rz -180 deg; joints [-156.028, -72.614, -46.56, 42.37, 37.077, -36.045]
  Call Extruder(206.06099)
  MoveL 5845 to (238.27, 42.22, 88.06) mm, rotated rx -180 ry 0 rz 180 deg; joints [-156.012, -72.645, -46.493, 42.423, 37.06, -36.102]
  MoveL 5846 to (238.27, 42.22, 88.06) mm, rotated rx -180 ry 0 rz 180 deg; joints [-156.012, -72.645, -46.493, 42.423, 37.06, -36.102]
  Call Extruder(206.21452)
  MoveL 5847 to (238.4, 42.44, 88.06) mm, rotated rx -180 ry 0 rz 180 deg; joints [-155.997, -72.674, -46.432, 42.472, 37.045, -36.154]
  MoveL 5848 to (238.4, 42.44, 88.06) mm, rotated rx -180 ry 0 rz 180 deg; joints [-155.997, -72.674, -46.432, 42.472, 37.045, -36.154]
  Call Extruder(206.42306)
  MoveL 5849 to (238.58, 42.75, 88.06) mm, rotated rx 180 ry 0 rz -180 deg; joints [-155.977, -72.713, -46.349, 42.539, 37.025, -36.225]
  MoveL 5850 to (238.58, 42.75, 88.06) mm, rotated rx 180 ry 0 rz -180 deg; joints [-155.977, -72.713, -46.349, 42.539, 37.025, -36.225]
  Call Extruder(206.63087)
  MoveL 5851 to (238.75, 43.06, 88.06) mm, rotated rx 180 ry 0 rz -180 deg; joints [-155.956, -72.752, -46.266, 42.606, 37.005, -36.297]
  MoveL 5852 to (238.75, 43.06, 88.06) mm, rotated rx 180 ry 0 rz -180 deg; joints [-155.956, -72.752, -46.266, 42.606, 37.005, -36.297]
  Call Extruder(206.81346)
  MoveL 5853 to (238.89, 43.33, 88.06) mm, rotated rx -180 ry 0 rz 180 deg; joints [-155.937, -72.786, -46.195, 42.665, 36.989, -36.359]
  MoveL 5854 to (238.89, 43.33, 88.06) mm, rotated rx -180 ry 0 rz 180 deg; joints [-155.937, -72.786, -46.195, 42.665, 36.989, -36.359]
  Call Extruder(206.97148)
  MoveL 5855 to (239, 43.58, 88.06) mm, rotated rx -180 ry 0 rz -180 deg; joints [-155.919, -72.813, -46.137, 42.717, 36.977, -36.413]
  MoveL 5856 to (239, 43.58, 88.06) mm, rotated rx -180 ry 0 rz -180 deg; joints [-155.919, -72.813, -46.137, 42.717, 36.977, -36.413]
  Call Extruder(207.12890)
  MoveL 5857 to (239.1, 43.83, 88.06) mm, rotated rx 180 ry 0 rz -180 deg; joints [-155.901, -72.841, -46.079, 42.769, 36.965, -36.467]
  MoveL 5858 to (239.1, 43.83, 88.06) mm, rotated rx 180 ry 0 rz -180 deg; joints [-155.901, -72.841, -46.079, 42.769, 36.965, -36.467]
  Call Extruder(207.31161)
  MoveL 5859 to (239.23, 44.12, 88.06) mm, rotated rx 180 ry 0 rz 180 deg; joints [-155.879, -72.872, -46.012, 42.829, 36.951, -36.53]
  MoveL 5860 to (239.23, 44.12, 88.06) mm, rotated rx 180 ry 0 rz 180 deg; joints [-155.879, -72.872, -46.012, 42.829, 36.951, -36.53]
  Call Extruder(207.49357)
  MoveL 5861 to (239.35, 44.42, 88.06) mm, rotated rx -180 ry 0 rz -180 deg; joints [-155.858, -72.904, -45.945, 42.89, 36.938, -36.593]
  MoveL 5862 to (239.35, 44.42, 88.06) mm, rotated rx -180 ry 0 rz -180 deg; joints [-155.858, -72.904, -45.945, 42.89, 36.938, -36.593]
  Call Extruder(207.64090)
  MoveL 5863 to (239.44, 44.66, 88.06) mm, rotated rx 180 ry 0 rz -180 deg; joints [-155.84, -72.929, -45.892, 42.939, 36.928, -36.644]
  MoveL 5864 to (239.44, 44.66, 88.06) mm, rotated rx 180 ry 0 rz -180 deg; joints [-155.84, -72.929, -45.892, 42.939, 36.928, -36.644]
  Call Extruder(207.75414)
  MoveL 5865 to (239.5, 44.85, 88.06) mm, rotated rx 180 ry 0 rz 180 deg; joints [-155.826, -72.947, -45.852, 42.977, 36.921, -36.683]
  MoveL 5866 to (239.5, 44.85, 88.06) mm, rotated rx 180 ry 0 rz 180 deg; joints [-155.826, -72.947, -45.852, 42.977, 36.921, -36.683]
  Call Extruder(207.86693)
  MoveL 5867 to (239.56, 45.03, 88.06) mm, rotated rx 180 ry 0 rz 180 deg; joints [-155.811, -72.966, -45.813, 43.015, 36.915, -36.721]
  MoveL 5868 to (239.56, 45.03, 88.06) mm, rotated rx 180 ry 0 rz 180 deg; joints [-155.811, -72.966, -45.813, 43.015, 36.915, -36.721]
  Call Extruder(207.97927)
  MoveL 5869 to (239.62, 45.22, 88.06) mm, rotated rx 180 ry 0 rz -180 deg; joints [-155.797, -72.984, -45.774, 43.053, 36.908, -36.76]
  MoveL 5870 to (239.62, 45.22, 88.06) mm, rotated rx 180 ry 0 rz -180 deg; joints [-155.797, -72.984, -45.774, 43.053, 36.908, -36.76]
  Call Extruder(208.09117)
  MoveL 5871 to (239.68, 45.41, 88.06) mm, rotated rx 180 ry 0 rz 180 deg; joints [-155.783, -73.003, -45.735, 43.091, 36.902, -36.799]
  MoveL 5872 to (239.68, 45.41, 88.06) mm, rotated rx 180 ry 0 rz 180 deg; joints [-155.783, -73.003, -45.735, 43.091, 36.902, -36.799]
  Call Extruder(208.21257)
  MoveL 5873 to (239.75, 45.62, 88.06) mm, rotated rx 180 ry 0 rz 180 deg; joints [-155.767, -73.023, -45.693, 43.132, 36.895, -36.841]
  MoveL 5874 to (239.75, 45.62, 88.06) mm, rotated rx 180 ry 0 rz 180 deg; joints [-155.767, -73.023, -45.693, 43.132, 36.895, -36.841]
  Call Extruder(208.34336)
  MoveL 5875 to (239.81, 45.84, 88.06) mm, rotated rx 180 ry 0 rz 180 deg; joints [-155.75, -73.044, -45.648, 43.177, 36.888, -36.887]
  MoveL 5876 to (239.81, 45.84, 88.06) mm, rotated rx 180 ry 0 rz 180 deg; joints [-155.75, -73.044, -45.648, 43.177, 36.888, -36.887]
  Call Extruder(208.47359)
  MoveL 5877 to (239.88, 46.06, 88.06) mm, rotated rx 180 ry 0 rz 180 deg; joints [-155.733, -73.065, -45.603, 43.221, 36.881, -36.932]
  MoveL 5878 to (239.88, 46.06, 88.06) mm, rotated rx 180 ry 0 rz 180 deg; joints [-155.733, -73.065, -45.603, 43.221, 36.881, -36.932]
  Call Extruder(208.60325)
  MoveL 5879 to (239.95, 46.29, 88.06) mm, rotated rx 180 ry 0 rz 180 deg; joints [-155.715, -73.087, -45.557, 43.266, 36.874, -36.978]
  MoveL 5880 to (239.95, 46.29, 88.06) mm, rotated rx 180 ry 0 rz 180 deg; joints [-155.715, -73.087, -45.557, 43.266, 36.874, -36.978]
  Call Extruder(208.73235)
  MoveL 5881 to (240.02, 46.51, 88.06) mm, rotated rx 180 ry 0 rz 180 deg; joints [-155.698, -73.108, -45.512, 43.311, 36.867, -37.024]
  MoveL 5882 to (240.02, 46.51, 88.06) mm, rotated rx 180 ry 0 rz 180 deg; joints [-155.698, -73.108, -45.512, 43.311, 36.867, -37.024]
  Call Extruder(208.84740)
  MoveL 5883 to (240.06, 46.72, 88.06) mm, rotated rx -180 ry 0 rz -180 deg; joints [-155.682, -73.125, -45.475, 43.35, 36.863, -37.063]
  MoveL 5884 to (240.06, 46.72, 88.06) mm, rotated rx -180 ry 0 rz -180 deg; joints [-155.682, -73.125, -45.475, 43.35, 36.863, -37.063]
  Call Extruder(208.96201)
  MoveL 5885 to (240.11, 46.92, 88.06) mm, rotated rx 180 ry 0 rz -180 deg; joints [-155.665, -73.143, -45.438, 43.39, 36.858, -37.103]
  MoveL 5886 to (240.11, 46.92, 88.06) mm, rotated rx 180 ry 0 rz -180 deg; joints [-155.665, -73.143, -45.438, 43.39, 36.858, -37.103]
  Call Extruder(209.07616)
  MoveL 5887 to (240.15, 47.12, 88.06) mm, rotated rx 180 ry 0 rz 180 deg; joints [-155.649, -73.16, -45.401, 43.43, 36.854, -37.143]
  MoveL 5888 to (240.15, 47.12, 88.06) mm, rotated rx 180 ry 0 rz 180 deg; joints [-155.649, -73.16, -45.401, 43.43, 36.854, -37.143]
  Call Extruder(209.18985)
  MoveL 5889 to (240.2, 47.33, 88.06) mm, rotated rx 180 ry 0 rz 180 deg; joints [-155.633, -73.178, -45.364, 43.469, 36.85, -37.182]
  MoveL 5890 to (240.2, 47.33, 88.06) mm, rotated rx 180 ry 0 rz 180 deg; joints [-155.633, -73.178, -45.364, 43.469, 36.85, -37.182]
  Call Extruder(209.31526)
  MoveL 5891 to (240.24, 47.55, 88.06) mm, rotated rx -180 ry 0 rz 180 deg; joints [-155.614, -73.197, -45.324, 43.513, 36.845, -37.226]
  MoveL 5892 to (240.24, 47.55, 88.06) mm, rotated rx -180 ry 0 rz 180 deg; joints [-155.614, -73.197, -45.324, 43.513, 36.845, -37.226]
  Call Extruder(209.45224)
  MoveL 5893 to (240.29, 47.8, 88.06) mm, rotated rx -180 ry 0 rz 180 deg; joints [-155.594, -73.218, -45.28, 43.561, 36.841, -37.274]
  MoveL 5894 to (240.29, 47.8, 88.06) mm, rotated rx -180 ry 0 rz 180 deg; joints [-155.594, -73.218, -45.28, 43.561, 36.841, -37.274]
  Call Extruder(209.58861)
  MoveL 5895 to (240.34, 48.05, 88.06) mm, rotated rx -180 ry 0 rz -180 deg; joints [-155.574, -73.238, -45.236, 43.609, 36.836, -37.322]
  MoveL 5896 to (240.34, 48.05, 88.06) mm, rotated rx -180 ry 0 rz -180 deg; joints [-155.574, -73.238, -45.236, 43.609, 36.836, -37.322]
  Call Extruder(209.72437)
  MoveL 5897 to (240.39, 48.3, 88.06) mm, rotated rx 180 ry 0 rz 180 deg; joints [-155.554, -73.259, -45.192, 43.657, 36.832, -37.37]
  MoveL 5898 to (240.39, 48.3, 88.06) mm, rotated rx 180 ry 0 rz 180 deg; joints [-155.554, -73.259, -45.192, 43.657, 36.832, -37.37]
  Call Extruder(209.85951)
  MoveL 5899 to (240.44, 48.55, 88.06) mm, rotated rx -180 ry 0 rz 180 deg; joints [-155.534, -73.28, -45.148, 43.705, 36.827, -37.418]
  MoveL 5900 to (240.44, 48.55, 88.06) mm, rotated rx -180 ry 0 rz 180 deg; joints [-155.534, -73.28, -45.148, 43.705, 36.827, -37.418]
  Call Extruder(209.99405)
  MoveL 5901 to (240.49, 48.8, 88.06) mm, rotated rx -180 ry 0 rz 180 deg; joints [-155.514, -73.301, -45.104, 43.753, 36.822, -37.466]
  MoveL 5902 to (240.49, 48.8, 88.06) mm, rotated rx -180 ry 0 rz 180 deg; joints [-155.514, -73.301, -45.104, 43.753, 36.822, -37.466]
  Call Extruder(210.12798)
  MoveL 5903 to (240.54, 49.05, 88.06) mm, rotated rx 180 ry 0 rz -180 deg; joints [-155.494, -73.321, -45.06, 43.801, 36.818, -37.514]
  MoveL 5904 to (240.54, 49.05, 88.06) mm, rotated rx 180 ry 0 rz -180 deg; joints [-155.494, -73.321, -45.06, 43.801, 36.818, -37.514]
  Call Extruder(210.27584)
  MoveL 5905 to (240.59, 49.33, 88.06) mm, rotated rx 180 ry 0 rz -180 deg; joints [-155.471, -73.344, -45.013, 43.854, 36.814, -37.567]
  MoveL 5906 to (240.59, 49.33, 88.06) mm, rotated rx 180 ry 0 rz -180 deg; joints [-155.471, -73.344, -45.013, 43.854, 36.814, -37.567]
  Call Extruder(210.43759)
  MoveL 5907 to (240.64, 49.63, 88.06) mm, rotated rx 180 ry 0 rz -180 deg; joints [-155.446, -73.368, -44.962, 43.912, 36.81, -37.625]
  MoveL 5908 to (240.64, 49.63, 88.06) mm, rotated rx 180 ry 0 rz -180 deg; joints [-155.446, -73.368, -44.962, 43.912, 36.81, -37.625]
  Call Extruder(210.59860)
  MoveL 5909 to (240.69, 49.94, 88.06) mm, rotated rx -180 ry 0 rz 180 deg; joints [-155.421, -73.392, -44.911, 43.97, 36.806, -37.683]
  MoveL 5910 to (240.69, 49.94, 88.06) mm, rotated rx -180 ry 0 rz 180 deg; joints [-155.421, -73.392, -44.911, 43.97, 36.806, -37.683]
  Call Extruder(210.75889)
  MoveL 5911 to (240.74, 50.24, 88.06) mm, rotated rx 180 ry 0 rz 180 deg; joints [-155.396, -73.416, -44.86, 44.028, 36.802, -37.74]
  MoveL 5912 to (240.74, 50.24, 88.06) mm, rotated rx 180 ry 0 rz 180 deg; joints [-155.396, -73.416, -44.86, 44.028, 36.802, -37.74]
  Call Extruder(210.91845)
  MoveL 5913 to (240.78, 50.55, 88.06) mm, rotated rx 180 ry 0 rz 180 deg; joints [-155.371, -73.44, -44.809, 44.087, 36.798, -37.798]
  MoveL 5914 to (240.78, 50.55, 88.06) mm, rotated rx 180 ry 0 rz 180 deg; joints [-155.371, -73.44, -44.809, 44.087, 36.798, -37.798]
  Call Extruder(211.07728)
  MoveL 5915 to (240.83, 50.86, 88.06) mm, rotated rx 180 ry 0 rz 180 deg; joints [-155.346, -73.465, -44.757, 44.145, 36.794, -37.856]
  MoveL 5916 to (240.83, 50.86, 88.06) mm, rotated rx 180 ry 0 rz 180 deg; joints [-155.346, -73.465, -44.757, 44.145, 36.794, -37.856]
  Call Extruder(211.25596)
  MoveL 5917 to (240.88, 51.2, 88.06) mm, rotated rx 180 ry 0 rz 180 deg; joints [-155.317, -73.491, -44.702, 44.21, 36.79, -37.92]
  MoveL 5918 to (240.88, 51.2, 88.06) mm, rotated rx 180 ry 0 rz 180 deg; joints [-155.317, -73.491, -44.702, 44.21, 36.79, -37.92]
  Call Extruder(211.45440)
  MoveL 5919 to (240.92, 51.59, 88.06) mm, rotated rx 180 ry 0 rz -180 deg; joints [-155.285, -73.52, -44.641, 44.283, 36.787, -37.992]
  MoveL 5920 to (240.92, 51.59, 88.06) mm, rotated rx 180 ry 0 rz -180 deg; joints [-155.285, -73.52, -44.641, 44.283, 36.787, -37.992]
  Call Extruder(211.65197)
  MoveL 5921 to (240.97, 51.98, 88.06) mm, rotated rx 180 ry 0 rz 180 deg; joints [-155.252, -73.549, -44.58, 44.355, 36.784, -38.064]
  MoveL 5922 to (240.97, 51.98, 88.06) mm, rotated rx 180 ry 0 rz 180 deg; joints [-155.252, -73.549, -44.58, 44.355, 36.784, -38.064]
  Call Extruder(211.84868)
  MoveL 5923 to (241.02, 52.36, 88.06) mm, rotated rx 180 ry 0 rz 180 deg; joints [-155.22, -73.578, -44.518, 44.428, 36.781, -38.135]
  MoveL 5924 to (241.02, 52.36, 88.06) mm, rotated rx 180 ry 0 rz 180 deg; joints [-155.22, -73.578, -44.518, 44.428, 36.781, -38.135]
  Call Extruder(212.04452)
  MoveL 5925 to (241.06, 52.75, 88.06) mm, rotated rx -180 ry 0 rz 180 deg; joints [-155.188, -73.607, -44.457, 44.5, 36.778, -38.207]
  MoveL 5926 to (241.06, 52.75, 88.06) mm, rotated rx -180 ry 0 rz 180 deg; joints [-155.188, -73.607, -44.457, 44.5, 36.778, -38.207]
  Call Extruder(212.33996)
  MoveL 5927 to (241.11, 53.34, 88.06) mm, rotated rx -180 ry 0 rz 180 deg; joints [-155.138, -73.648, -44.37, 44.609, 36.776, -38.313]
  MoveL 5928 to (241.11, 53.34, 88.06) mm, rotated rx -180 ry 0 rz 180 deg; joints [-155.138, -73.648, -44.37, 44.609, 36.776, -38.313]
  Call Extruder(212.63406)
  MoveL 5929 to (241.16, 53.93, 88.06) mm, rotated rx 180 ry 0 rz 180 deg; joints [-155.088, -73.689, -44.283, 44.718, 36.775, -38.419]
  MoveL 5930 to (241.16, 53.93, 88.06) mm, rotated rx 180 ry 0 rz 180 deg; joints [-155.088, -73.689, -44.283, 44.718, 36.775, -38.419]
  Call Extruder(212.92684)
  MoveL 5931 to (241.2, 54.52, 88.06) mm, rotated rx -180 ry 0 rz -180 deg; joints [-155.038, -73.731, -44.195, 44.826, 36.773, -38.526]
  MoveL 5932 to (241.2, 54.52, 88.06) mm, rotated rx -180 ry 0 rz -180 deg; joints [-155.038, -73.731, -44.195, 44.826, 36.773, -38.526]
  Call Extruder(213.50029)
  MoveL 5933 to (241.25, 55.68, 88.06) mm, rotated rx -180 ry 0 rz 180 deg; joints [-154.938, -73.807, -44.034, 45.037, 36.775, -38.731]
  MoveL 5934 to (241.25, 55.68, 88.06) mm, rotated rx -180 ry 0 rz 180 deg; joints [-154.938, -73.807, -44.034, 45.037, 36.775, -38.731]
  Call Extruder(214.21412)
  MoveL 5935 to (241.29, 57.14, 88.06) mm, rotated rx -180 ry 0 rz -180 deg; joints [-154.812, -73.901, -43.837, 45.299, 36.781, -38.985]
  Call Extruder(256.27901)
  MoveL 5936 to (241.29, 142.86, 88.06) mm, rotated rx 180 ry 0 rz 180 deg; joints [-147.778, -80.766, -29.631, 61.058, 37.538, -55.109]
  Call Extruder(256.70743)
  MoveL 5937 to (241.27, 143.73, 88.06) mm, rotated rx -180 ry 0 rz 180 deg; joints [-147.711, -80.855, -29.45, 61.226, 37.549, -55.291]
  MoveL 5938 to (241.27, 143.73, 88.06) mm, rotated rx -180 ry 0 rz 180 deg; joints [-147.711, -80.855, -29.45, 61.226, 37.549, -55.291]
  Call Extruder(257.28088)
  MoveL 5939 to (241.22, 144.9, 88.06) mm, rotated rx -180 ry 0 rz 180 deg; joints [-147.62, -80.971, -29.215, 61.447, 37.567, -55.53]
  MoveL 5940 to (241.22, 144.9, 88.06) mm, rotated rx -180 ry 0 rz 180 deg; joints [-147.62, -80.971, -29.215, 61.447, 37.567, -55.53]
  Call Extruder(257.71522)
  MoveL 5941 to (241.18, 145.77, 88.06) mm, rotated rx 180 ry 0 rz 180 deg; joints [-147.551, -81.056, -29.041, 61.612, 37.582, -55.708]
  MoveL 5942 to (241.18, 145.77, 88.06) mm, rotated rx 180 ry 0 rz 180 deg; joints [-147.551, -81.056, -29.041, 61.612, 37.582, -55.708]
  Call Extruder(258.00933)
  MoveL 5943 to (241.13, 146.36, 88.06) mm, rotated rx -180 ry 0 rz -180 deg; joints [-147.504, -81.111, -28.929, 61.721, 37.594, -55.825]
  MoveL 5944 to (241.13, 146.36, 88.06) mm, rotated rx -180 ry 0 rz -180 deg; joints [-147.504, -81.111, -28.929, 61.721, 37.594, -55.825]
  Call Extruder(258.30477)
  MoveL 5945 to (241.09, 146.95, 88.06) mm, rotated rx 180 ry 0 rz 180 deg; joints [-147.457, -81.167, -28.816, 61.83, 37.606, -55.942]
  MoveL 5946 to (241.09, 146.95, 88.06) mm, rotated rx 180 ry 0 rz 180 deg; joints [-147.457, -81.167, -28.816, 61.83, 37.606, -55.942]
  Call Extruder(258.55103)
  MoveL 5947 to (241.04, 147.44, 88.06) mm, rotated rx 180 ry 0 rz 180 deg; joints [-147.417, -81.212, -28.725, 61.919, 37.616, -56.038]
  MoveL 5948 to (241.04, 147.44, 88.06) mm, rotated rx 180 ry 0 rz 180 deg; joints [-147.417, -81.212, -28.725, 61.919, 37.616, -56.038]
  Call Extruder(258.74773)
  MoveL 5949 to (240.99, 147.83, 88.06) mm, rotated rx -180 ry 0 rz -180 deg; joints [-147.386, -81.246, -28.655, 61.988, 37.626, -56.111]
  MoveL 5950 to (240.99, 147.83, 88.06) mm, rotated rx -180 ry 0 rz -180 deg; joints [-147.386, -81.246, -28.655, 61.988, 37.626, -56.111]
  Call Extruder(258.94530)
  MoveL 5951 to (240.95, 148.22, 88.06) mm, rotated rx 180 ry 0 rz 180 deg; joints [-147.354, -81.281, -28.586, 62.057, 37.636, -56.185]
  MoveL 5952 to (240.95, 148.22, 88.06) mm, rotated rx 180 ry 0 rz 180 deg; joints [-147.354, -81.281, -28.586, 62.057, 37.636, -56.185]
  Call Extruder(259.14375)
  MoveL 5953 to (240.9, 148.6, 88.06) mm, rotated rx -180 ry 0 rz -180 deg; joints [-147.322, -81.315, -28.516, 62.127, 37.645, -56.259]
  MoveL 5954 to (240.9, 148.6, 88.06) mm, rotated rx -180 ry 0 rz -180 deg; joints [-147.322, -81.315, -28.516, 62.127, 37.645, -56.259]
  Call Extruder(259.34306)
  MoveL 5955 to (240.86, 148.99, 88.06) mm, rotated rx 180 ry 0 rz -180 deg; joints [-147.291, -81.349, -28.446, 62.196, 37.655, -56.333]
  MoveL 5956 to (240.86, 148.99, 88.06) mm, rotated rx 180 ry 0 rz -180 deg; joints [-147.291, -81.349, -28.446, 62.196, 37.655, -56.333]
  Call Extruder(259.50189)
  MoveL 5957 to (240.81, 149.3, 88.06) mm, rotated rx -180 ry 0 rz 180 deg; joints [-147.265, -81.375, -28.395, 62.249, 37.664, -56.389]
  MoveL 5958 to (240.81, 149.3, 88.06) mm, rotated rx -180 ry 0 rz 180 deg; joints [-147.265, -81.375, -28.395, 62.249, 37.664, -56.389]
  Call Extruder(259.66145)
  MoveL 5959 to (240.76, 149.6, 88.06) mm, rotated rx 180 ry 0 rz 180 deg; joints [-147.24, -81.4, -28.343, 62.302, 37.673, -56.445]
  MoveL 5960 to (240.76, 149.6, 88.06) mm, rotated rx 180 ry 0 rz 180 deg; joints [-147.24, -81.4, -28.343, 62.302, 37.673, -56.445]
  Call Extruder(259.82174)
  MoveL 5961 to (240.71, 149.91, 88.06) mm, rotated rx -180 ry 0 rz 180 deg; joints [-147.214, -81.425, -28.292, 62.355, 37.683, -56.501]
  MoveL 5962 to (240.71, 149.91, 88.06) mm, rotated rx -180 ry 0 rz 180 deg; joints [-147.214, -81.425, -28.292, 62.355, 37.683, -56.501]
  Call Extruder(259.98276)
  MoveL 5963 to (240.66, 150.21, 88.06) mm, rotated rx -180 ry 0 rz 180 deg; joints [-147.189, -81.451, -28.241, 62.407, 37.692, -56.557]
  MoveL 5964 to (240.66, 150.21, 88.06) mm, rotated rx -180 ry 0 rz 180 deg; joints [-147.189, -81.451, -28.241, 62.407, 37.692, -56.557]
  Call Extruder(260.14450)
  MoveL 5965 to (240.61, 150.52, 88.06) mm, rotated rx 180 ry 0 rz 180 deg; joints [-147.163, -81.476, -28.189, 62.46, 37.701, -56.613]
  MoveL 5966 to (240.61, 150.52, 88.06) mm, rotated rx 180 ry 0 rz 180 deg; joints [-147.163, -81.476, -28.189, 62.46, 37.701, -56.613]
  Call Extruder(260.30697)
  MoveL 5967 to (240.56, 150.83, 88.06) mm, rotated rx 180 ry 0 rz -180 deg; joints [-147.138, -81.502, -28.137, 62.513, 37.71, -56.669]
  MoveL 5968 to (240.56, 150.83, 88.06) mm, rotated rx 180 ry 0 rz -180 deg; joints [-147.138, -81.502, -28.137, 62.513, 37.71, -56.669]
  Call Extruder(260.44090)
  MoveL 5969 to (240.52, 151.07, 88.06) mm, rotated rx -180 ry 0 rz 180 deg; joints [-147.117, -81.521, -28.098, 62.555, 37.719, -56.713]
  MoveL 5970 to (240.52, 151.07, 88.06) mm, rotated rx -180 ry 0 rz 180 deg; joints [-147.117, -81.521, -28.098, 62.555, 37.719, -56.713]
  Call Extruder(260.57544)
  MoveL 5971 to (240.47, 151.32, 88.06) mm, rotated rx -180 ry 0 rz -180 deg; joints [-147.095, -81.54, -28.06, 62.597, 37.727, -56.757]
  MoveL 5972 to (240.47, 151.32, 88.06) mm, rotated rx -180 ry 0 rz -180 deg; joints [-147.095, -81.54, -28.06, 62.597, 37.727, -56.757]
  Call Extruder(260.71058)
  MoveL 5973 to (240.42, 151.57, 88.06) mm, rotated rx -180 ry 0 rz 180 deg; joints [-147.074, -81.559, -28.021, 62.638, 37.736, -56.8]
  MoveL 5974 to (240.42, 151.57, 88.06) mm, rotated rx -180 ry 0 rz 180 deg; joints [-147.074, -81.559, -28.021, 62.638, 37.736, -56.8]
  Call Extruder(260.84634)
  MoveL 5975 to (240.37, 151.82, 88.06) mm, rotated rx 180 ry 0 rz -180 deg; joints [-147.053, -81.578, -27.982, 62.68, 37.745, -56.844]
  MoveL 5976 to (240.37, 151.82, 88.06) mm, rotated rx 180 ry 0 rz -180 deg; joints [-147.053, -81.578, -27.982, 62.68, 37.745, -56.844]
  Call Extruder(260.98271)
  MoveL 5977 to (240.32, 152.07, 88.06) mm, rotated rx 180 ry 0 rz 180 deg; joints [-147.032, -81.597, -27.943, 62.721, 37.754, -56.887]
  MoveL 5978 to (240.32, 152.07, 88.06) mm, rotated rx 180 ry 0 rz 180 deg; joints [-147.032, -81.597, -27.943, 62.721, 37.754, -56.887]
  Call Extruder(261.11969)
  MoveL 5979 to (240.27, 152.32, 88.06) mm, rotated rx 180 ry 0 rz 180 deg; joints [-147.011, -81.617, -27.904, 62.763, 37.762, -56.931]
  MoveL 5980 to (240.27, 152.32, 88.06) mm, rotated rx 180 ry 0 rz 180 deg; joints [-147.011, -81.617, -27.904, 62.763, 37.762, -56.931]
  Call Extruder(261.25727)
  MoveL 5981 to (240.22, 152.57, 88.06) mm, rotated rx -180 ry 0 rz 180 deg; joints [-146.989, -81.636, -27.865, 62.804, 37.771, -56.975]
  MoveL 5982 to (240.22, 152.57, 88.06) mm, rotated rx -180 ry 0 rz 180 deg; joints [-146.989, -81.636, -27.865, 62.804, 37.771, -56.975]
  Call Extruder(261.37097)
  MoveL 5983 to (240.17, 152.77, 88.06) mm, rotated rx 180 ry 0 rz 180 deg; joints [-146.972, -81.651, -27.834, 62.838, 37.779, -57.01]
  MoveL 5984 to (240.17, 152.77, 88.06) mm, rotated rx 180 ry 0 rz 180 deg; joints [-146.972, -81.651, -27.834, 62.838, 37.779, -57.01]
  Call Extruder(261.48512)
  MoveL 5985 to (240.13, 152.98, 88.06) mm, rotated rx -180 ry 0 rz -180 deg; joints [-146.954, -81.666, -27.803, 62.872, 37.786, -57.045]
  MoveL 5986 to (240.13, 152.98, 88.06) mm, rotated rx -180 ry 0 rz -180 deg; joints [-146.954, -81.666, -27.803, 62.872, 37.786, -57.045]
  Call Extruder(261.59972)
  MoveL 5987 to (240.08, 153.18, 88.06) mm, rotated rx 180 ry 0 rz 180 deg; joints [-146.937, -81.681, -27.773, 62.905, 37.794, -57.08]
  MoveL 5988 to (240.08, 153.18, 88.06) mm, rotated rx 180 ry 0 rz 180 deg; joints [-146.937, -81.681, -27.773, 62.905, 37.794, -57.08]
  Call Extruder(261.71478)
  MoveL 5989 to (240.04, 153.39, 88.06) mm, rotated rx 180 ry 0 rz -180 deg; joints [-146.919, -81.697, -27.742, 62.939, 37.801, -57.115]
  MoveL 5990 to (240.04, 153.39, 88.06) mm, rotated rx 180 ry 0 rz -180 deg; joints [-146.919, -81.697, -27.742, 62.939, 37.801, -57.115]
  Call Extruder(261.83700)
  MoveL 5991 to (239.98, 153.6, 88.06) mm, rotated rx 180 ry 0 rz 180 deg; joints [-146.9, -81.711, -27.712, 62.972, 37.81, -57.149]
  MoveL 5992 to (239.98, 153.6, 88.06) mm, rotated rx 180 ry 0 rz 180 deg; joints [-146.9, -81.711, -27.712, 62.972, 37.81, -57.149]
  Call Extruder(261.96666)
